  [311] = {x=105.115163, y=10.552736, z=54.518881, rx=0.000471, ry=-77.672976, rz=0.000213, shoulder=lefty, elbow=epositive, wrist=wpositive, fatherId=frmaster[1]}
  [312] = {x=103.355897, y=10.008134, z=58.376297, rx=0.003948, ry=-79.793029, rz=0.003471, shoulder=lefty, elbow=epositive, wrist=wpositive, fatherId=frmaster[1]}
  [313] = {x=101.174698, y=9.463298, z=62.618231, rx=-0.002344, ry=-82.1673, rz=-0.001686, shoulder=lefty, elbow=epositive, wrist=wpositive, fatherId=frmaster[1]}
  [314] = {x=98.49876, y=8.920808, z=67.239802, rx=-0.00454, ry=-84.819695, rz=-0.004128, shoulder=lefty, elbow=epositive, wrist=wpositive, fatherId=frmaster[1]}
  [315] = {x=95.239995, y=8.372547, z=72.223013, rx=0.011592, ry=-87.766502, rz=0.011331, shoulder=lefty, elbow=epositive, wrist=wpositive, fatherId=frmaster[1]}
  [316] = {x=93.405559, y=8.100927, z=74.780335, rx=-0.033898, ry=-89.319085, rz=-0.033723, shoulder=lefty, elbow=epositive, wrist=wpositive, fatherId=frmaster[1]}
  [317] = {x=91.396985, y=7.822504, z=77.414063, rx=-0.028938, ry=-90.956699, rz=-0.029283, shoulder=lefty, elbow=epositive, wrist=wpositive, fatherId=frmaster[1]}
  [318] = {x=89.185601, y=7.550471, z=80.130199, rx=0.005621, ry=-92.678971, rz=0.005427, shoulder=lefty, elbow=epositive, wrist=wpositive, fatherId=frmaster[1]}
  [319] = {x=86.774878, y=7.274773, z=82.909129, rx=0.003041, ry=-94.483485, rz=0.003791, shoulder=lefty, elbow=epositive, wrist=wpositive, fatherId=frmaster[1]}
  [320] = {x=84.156667, y=6.996406, z=85.721464, rx=-0.004918, ry=-96.374138, rz=-0.004959, shoulder=lefty, elbow=epositive, wrist=wpositive, fatherId=frmaster[1]}
  [321] = {x=81.287604, y=6.727029, z=88.5933, rx=0.003959, ry=-98.361433, rz=0.003574, shoulder=lefty, elbow=epositive, wrist=wpositive, fatherId=frmaster[1]}
  [322] = {x=79.766548, y=6.586584, z=90.039185, rx=0.000425, ry=-99.39159, rz=0.000719, shoulder=lefty, elbow=epositive, wrist=wpositive, fatherId=frmaster[1]}
  [323] = {x=76.689148, y=6.449037, z=92.743901, rx=-0.000115, ry=-101.368846, rz=-0.000541, shoulder=lefty, elbow=epositive, wrist=wpositive, fatherId=frmaster[1]}
  [324] = {x=72.711608, y=6.313912, z=95.955052, rx=0.002122, ry=-103.831925, rz=0.001993, shoulder=lefty, elbow=epositive, wrist=wpositive, fatherId=frmaster[1]}
  [325] = {x=68.637625, y=6.172358, z=98.971235, rx=-0.001983, ry=-106.275746, rz=-0.001913, shoulder=lefty, elbow=epositive, wrist=wpositive, fatherId=frmaster[1]}
  [326] = {x=64.204516, y=6.039868, z=101.957261, rx=0.000455, ry=-108.850801, rz=0.000254, shoulder=lefty, elbow=epositive, wrist=wpositive, fatherId=frmaster[1]}
  [327] = {x=59.531454, y=5.903167, z=104.808277, rx=-0.001203, ry=-111.487024, rz=-0.000792, shoulder=lefty, elbow=epositive, wrist=wpositive, fatherId=frmaster[1]}
  [328] = {x=54.601522, y=5.770946, z=107.502565, rx=0.000365, ry=-114.193934, rz=0.000646, shoulder=lefty, elbow=epositive, wrist=wpositive, fatherId=frmaster[1]}
  [329] = {x=49.396662, y=5.639217, z=110.0302, rx=0.001439, ry=-116.981093, rz=0.001954, shoulder=lefty, elbow=epositive, wrist=wpositive, fatherId=frmaster[1]}
  [330] = {x=43.905536, y=5.503752, z=112.367074, rx=0.001098, ry=-119.853038, rz=0.000658, shoulder=lefty, elbow=epositive, wrist=wpositive, fatherId=frmaster[1]}
  [331] = {x=38.132318, y=5.363596, z=114.489668, rx=-0.000754, ry=-122.812896, rz=-0.000603, shoulder=lefty, elbow=epositive, wrist=wpositive, fatherId=frmaster[1]}
  [332] = {x=34.633497, y=4.830797, z=115.697094, rx=-0.000999, ry=-124.728621, rz=-0.001121, shoulder=lefty, elbow=epositive, wrist=wpositive, fatherId=frmaster[1]}
  [333] = {x=32.195231, y=4.70506, z=116.424337, rx=-0.000117, ry=-125.974891, rz=-0.000379, shoulder=lefty, elbow=epositive, wrist=wpositive, fatherId=frmaster[1]}
  [334] = {x=28.076069, y=4.572613, z=117.507648, rx=0.000442, ry=-128.036025, rz=0.000186, shoulder=lefty, elbow=epositive, wrist=wpositive, fatherId=frmaster[1]}
  [335] = {x=25.057832, y=4.509903, z=118.201438, rx=0.000783, ry=-129.528131, rz=0.00073, shoulder=lefty, elbow=epositive, wrist=wpositive, fatherId=frmaster[1]}
  [336] = {x=21.435467, y=4.448246, z=118.91733, rx=0.000494, ry=-131.301627, rz=0.000656, shoulder=lefty, elbow=epositive, wrist=wpositive, fatherId=frmaster[1]}
  [337] = {x=17.185232, y=4.383492, z=119.614102, rx=0.000155, ry=-133.367865, rz=-0.000541, shoulder=lefty, elbow=epositive, wrist=wpositive, fatherId=frmaster[1]}
  [338] = {x=12.286771, y=4.319735, z=120.224792, rx=-0.000552, ry=-135.732916, rz=-0.00113, shoulder=lefty, elbow=epositive, wrist=wpositive, fatherId=frmaster[1]}
  [339] = {x=6.745577, y=4.261009, z=120.666296, rx=0.000441, ry=-138.391097, rz=-0.000116, shoulder=lefty, elbow=epositive, wrist=wpositive, fatherId=frmaster[1]}
  [340] = {x=0.626957, y=4.196667, z=120.856505, rx=-0.000387, ry=-141.317793, rz=-0.001039, shoulder=lefty, elbow=epositive, wrist=wpositive, fatherId=frmaster[1]}
  [341] = {x=-2.621994, y=4.16578, z=120.834592, rx=-0.00037, ry=-142.86837, rz=-0.000772, shoulder=lefty, elbow=epositive, wrist=wpositive, fatherId=frmaster[1]}
  [342] = {x=-8.220207, y=4.074828, z=120.570259, rx=0.000153, ry=-145.562099, rz=-0.00037, shoulder=lefty, elbow=epositive, wrist=wpositive, fatherId=frmaster[1]}
  [343] = {x=-12.173458, y=3.969382, z=120.234965, rx=-0.000075, ry=-147.496461, rz=0.000392, shoulder=lefty, elbow=epositive, wrist=wpositive, fatherId=frmaster[1]}
  [344] = {x=-16.022992, y=3.85518, z=119.762733, rx=0.000192, ry=-149.390807, rz=-0.000615, shoulder=lefty, elbow=epositive, wrist=wpositive, fatherId=frmaster[1]}
  [345] = {x=-19.771417, y=3.747011, z=119.182824, rx=0.000374, ry=-151.245321, rz=0.000006, shoulder=lefty, elbow=epositive, wrist=wpositive, fatherId=frmaster[1]}
  [346] = {x=-23.423427, y=3.639804, z=118.496959, rx=0.000566, ry=-153.06052, rz=0.000355, shoulder=lefty, elbow=epositive, wrist=wpositive, fatherId=frmaster[1]}
  [347] = {x=-27.437918, y=3.551048, z=117.608317, rx=0.000174, ry=-155.071656, rz=0.000909, shoulder=lefty, elbow=epositive, wrist=wpositive, fatherId=frmaster[1]}
  [348] = {x=-31.369091, y=3.453416, z=116.586239, rx=-0.000044, ry=-157.059735, rz=-0.000033, shoulder=lefty, elbow=epositive, wrist=wpositive, fatherId=frmaster[1]}
  [349] = {x=-35.226903, y=3.369271, z=115.441477, rx=0.000359, ry=-159.027084, rz=0.000287, shoulder=lefty, elbow=epositive, wrist=wpositive, fatherId=frmaster[1]}
  [350] = {x=-39.002937, y=3.277168, z=114.177394, rx=-0.000265, ry=-160.976303, rz=-0.000033, shoulder=lefty, elbow=epositive, wrist=wpositive, fatherId=frmaster[1]}
  [351] = {x=-43.085326, y=3.21008, z=112.652085, rx=-0.000248, ry=-163.110961, rz=0.000271, shoulder=lefty, elbow=epositive, wrist=wpositive, fatherId=frmaster[1]}
  [352] = {x=-47.122027, y=3.142962, z=110.968346, rx=0.000202, ry=-165.252195, rz=0.000493, shoulder=lefty, elbow=epositive, wrist=wpositive, fatherId=frmaster[1]}
  [353] = {x=-51.112902, y=3.070675, z=109.124081, rx=-0.00013, ry=-167.405313, rz=-0.000632, shoulder=lefty, elbow=epositive, wrist=wpositive, fatherId=frmaster[1]}
  [354] = {x=-54.974323, y=3.001944, z=107.153098, rx=0.000016, ry=-169.528533, rz=-0.000202, shoulder=lefty, elbow=epositive, wrist=wpositive, fatherId=frmaster[1]}
  [355] = {x=-59.390551, y=2.918741, z=104.602883, rx=0.000164, ry=-172.082376, rz=0.000136, shoulder=lefty, elbow=epositive, wrist=wpositive, fatherId=frmaster[1]}
  [356] = {x=-62.947412, y=2.832964, z=102.322113, rx=-0.000195, ry=-174.220706, rz=-0.000037, shoulder=lefty, elbow=epositive, wrist=wpositive, fatherId=frmaster[1]}
  [357] = {x=-62.947085, y=2.832936, z=112.317767, rx=-0.000211, ry=-174.22099, rz=0.00026, shoulder=lefty, elbow=epositive, wrist=wpositive, fatherId=frmaster[1]}
  [358] = {x=-58.458944, y=2.836341, z=156.681093, rx=0.000113, ry=-174.221159, rz=-0.000294, shoulder=lefty, elbow=epositive, wrist=wpositive, fatherId=frmaster[1]}
  [359] = {x=-18.612921, y=-20.076149, z=152.745219, rx=0.000402, ry=-174.056296, rz=-89.999944, shoulder=lefty, elbow=epositive, wrist=wpositive, fatherId=frmaster[1]}
  [360] = {x=-23.229929, y=-20.077149, z=108.388484, rx=-0.000285, ry=-174.056902, rz=-89.9999, shoulder=lefty, elbow=epositive, wrist=wpositive, fatherId=frmaster[1]}
  [361] = {x=-23.230934, y=-20.076541, z=98.391781, rx=0.000061, ry=-174.055786, rz=-89.999911, shoulder=lefty, elbow=epositive, wrist=wpositive, fatherId=frmaster[1]}
  [362] = {x=-19.340255, y=-20.472646, z=99.305974, rx=0.000015, ry=-171.571206, rz=-89.999811, shoulder=lefty, elbow=epositive, wrist=wpositive, fatherId=frmaster[1]}
  [363] = {x=-14.467347, y=-20.9313, z=100.19443, rx=179.999772, ry=-11.415156, rz=89.999471, shoulder=lefty, elbow=epositive, wrist=wpositive, fatherId=frmaster[1]}
  [364] = {x=-10.841793, y=-21.30275, z=100.675983, rx=-179.999737, ry=-13.600464, rz=89.99978, shoulder=lefty, elbow=epositive, wrist=wpositive, fatherId=frmaster[1]}
  [365] = {x=-6.648279, y=-21.675563, z=101.059651, rx=-0.000485, ry=-163.903958, rz=-89.999942, shoulder=lefty, elbow=epositive, wrist=wpositive, fatherId=frmaster[1]}
  [366] = {x=-3.944084, y=-21.97213, z=101.205494, rx=-179.999845, ry=-17.692348, rz=89.99981, shoulder=lefty, elbow=epositive, wrist=wpositive, fatherId=frmaster[1]}
  [367] = {x=-1.035961, y=-22.266805, z=101.281579, rx=0.000164, ry=-160.596349, rz=-89.999518, shoulder=lefty, elbow=epositive, wrist=wpositive, fatherId=frmaster[1]}
  [368] = {x=2.075668, y=-22.563936, z=101.263735, rx=-0.000431, ry=-158.771258, rz=-89.999398, shoulder=lefty, elbow=epositive, wrist=wpositive, fatherId=frmaster[1]}
  [369] = {x=5.374886, y=-22.856509, z=101.139982, rx=-0.00019, ry=-156.835849, rz=-89.999944, shoulder=lefty, elbow=epositive, wrist=wpositive, fatherId=frmaster[1]}
  [370] = {x=8.11646, y=-23.167098, z=100.948464, rx=179.999554, ry=-24.769598, rz=89.999348, shoulder=lefty, elbow=epositive, wrist=wpositive, fatherId=frmaster[1]}
  [371] = {x=10.839252, y=-23.473657, z=100.680376, rx=-179.999737, ry=-26.365625, rz=89.9993, shoulder=lefty, elbow=epositive, wrist=wpositive, fatherId=frmaster[1]}
  [372] = {x=14.340968, y=-24.085732, z=100.215497, rx=-179.999799, ry=-28.466933, rz=89.999508, shoulder=lefty, elbow=epositive, wrist=wpositive, fatherId=frmaster[1]}
  [373] = {x=17.063864, y=-24.631859, z=99.772139, rx=0.000249, ry=-149.886158, rz=-89.998887, shoulder=lefty, elbow=epositive, wrist=wpositive, fatherId=frmaster[1]}
  [374] = {x=19.727245, y=-25.186439, z=99.251868, rx=0.00024, ry=-148.268713, rz=-89.999973, shoulder=lefty, elbow=epositive, wrist=wpositive, fatherId=frmaster[1]}
  [375] = {x=23.493787, y=-26.015884, z=98.378332, rx=0.000126, ry=-145.960874, rz=-89.999685, shoulder=lefty, elbow=epositive, wrist=wpositive, fatherId=frmaster[1]}
  [376] = {x=27.151839, y=-26.844047, z=97.374762, rx=0.000396, ry=-143.695243, rz=-89.999786, shoulder=lefty, elbow=epositive, wrist=wpositive, fatherId=frmaster[1]}
  [377] = {x=30.702102, y=-27.677126, z=96.257879, rx=-0.001043, ry=-141.467559, rz=-89.999909, shoulder=lefty, elbow=epositive, wrist=wpositive, fatherId=frmaster[1]}
  [378] = {x=34.151197, y=-28.501632, z=95.007831, rx=0.000632, ry=-139.275172, rz=-89.999692, shoulder=lefty, elbow=epositive, wrist=wpositive, fatherId=frmaster[1]}
  [379] = {x=38.358157, y=-29.614839, z=93.291762, rx=179.999103, ry=-43.445668, rz=89.999456, shoulder=lefty, elbow=epositive, wrist=wpositive, fatherId=frmaster[1]}
  [380] = {x=40.816315, y=-30.16554, z=92.181405, rx=0.00035, ry=-134.95198, rz=-89.999842, shoulder=lefty, elbow=epositive, wrist=wpositive, fatherId=frmaster[1]}
  [381] = {x=43.623166, y=-30.723277, z=90.828073, rx=179.999263, ry=-46.887972, rz=89.999132, shoulder=lefty, elbow=epositive, wrist=wpositive, fatherId=frmaster[1]}
  [382] = {x=46.461035, y=-31.27399, z=89.349237, rx=0.000666, ry=-131.224555, rz=-89.999069, shoulder=lefty, elbow=epositive, wrist=wpositive, fatherId=frmaster[1]}
  [383] = {x=49.52499, y=-31.829878, z=87.61862, rx=0.000856, ry=-129.161053, rz=-89.998786, shoulder=lefty, elbow=epositive, wrist=wpositive, fatherId=frmaster[1]}
  [384] = {x=52.824587, y=-32.39186, z=85.592884, rx=-0.000376, ry=-126.896424, rz=-89.999824, shoulder=lefty, elbow=epositive, wrist=wpositive, fatherId=frmaster[1]}
  [385] = {x=56.368122, y=-32.945099, z=83.214974, rx=179.999887, ry=-55.592047, rz=89.99993, shoulder=lefty, elbow=epositive, wrist=wpositive, fatherId=frmaster[1]}
  [386] = {x=59.982794, y=-33.501646, z=80.56291, rx=0.000356, ry=-121.795353, rz=-89.999372, shoulder=lefty, elbow=epositive, wrist=wpositive, fatherId=frmaster[1]}
  [387] = {x=63.860131, y=-34.057469, z=77.43317, rx=0.001113, ry=-118.892986, rz=-89.998492, shoulder=lefty, elbow=epositive, wrist=wpositive, fatherId=frmaster[1]}
  [388] = {x=65.894571, y=-34.341079, z=75.654242, rx=179.999036, ry=-62.672719, rz=89.998766, shoulder=lefty, elbow=epositive, wrist=wpositive, fatherId=frmaster[1]}
  [389] = {x=67.978967, y=-34.617239, z=73.736742, rx=0.000688, ry=-115.679952, rz=-89.998265, shoulder=lefty, elbow=epositive, wrist=wpositive, fatherId=frmaster[1]}
  [390] = {x=70.113955, y=-34.895869, z=71.65174, rx=179.999274, ry=-66.045856, rz=89.999704, shoulder=lefty, elbow=epositive, wrist=wpositive, fatherId=frmaster[1]}
  [391] = {x=72.277536, y=-35.178962, z=69.406219, rx=179.998605, ry=-67.852148, rz=89.998988, shoulder=lefty, elbow=epositive, wrist=wpositive, fatherId=frmaster[1]}
  [392] = {x=74.376116, y=-35.45348, z=67.085303, rx=179.999869, ry=-69.662949, rz=89.999758, shoulder=lefty, elbow=epositive, wrist=wpositive, fatherId=frmaster[1]}
  [393] = {x=76.513977, y=-35.730157, z=64.566903, rx=0.000592, ry=-108.424559, rz=-89.999536, shoulder=lefty, elbow=epositive, wrist=wpositive, fatherId=frmaster[1]}
  [394] = {x=78.679667, y=-36.009316, z=61.843135, rx=0.001385, ry=-106.410069, rz=-89.998392, shoulder=lefty, elbow=epositive, wrist=wpositive, fatherId=frmaster[1]}
  [395] = {x=80.846119, y=-36.288822, z=58.903263, rx=0.000878, ry=-104.297201, rz=-89.999128, shoulder=lefty, elbow=epositive, wrist=wpositive, fatherId=frmaster[1]}
  [396] = {x=82.995135, y=-36.570009, z=55.747917, rx=179.999305, ry=-77.907489, rz=89.999806, shoulder=lefty, elbow=epositive, wrist=wpositive, fatherId=frmaster[1]}
  [397] = {x=85.094465, y=-36.847128, z=52.391805, rx=0.001232, ry=-99.802552, rz=-89.998506, shoulder=lefty, elbow=epositive, wrist=wpositive, fatherId=frmaster[1]}
  [398] = {x=87.124675, y=-37.127203, z=48.843094, rx=0.000325, ry=-97.44439, rz=-89.999996, shoulder=lefty, elbow=epositive, wrist=wpositive, fatherId=frmaster[1]}
  [399] = {x=89.220179, y=-37.40856, z=44.781627, rx=179.996062, ry=-85.19367, rz=89.995853, shoulder=lefty, elbow=epositive, wrist=wpositive, fatherId=frmaster[1]}
  [400] = {x=90.407375, y=-37.548857, z=42.270351, rx=0.000347, ry=-93.204424, rz=-89.999876, shoulder=lefty, elbow=epositive, wrist=wpositive, fatherId=frmaster[1]}
  [401] = {x=91.449184, y=-37.685314, z=39.897994, rx=179.994643, ry=-88.288606, rz=89.994157, shoulder=lefty, elbow=epositive, wrist=wpositive, fatherId=frmaster[1]}
  [402] = {x=93.126378, y=-37.965093, z=35.654137, rx=-0.009346, ry=-89.071193, rz=-90.008547, shoulder=lefty, elbow=epositive, wrist=wpositive, fatherId=frmaster[1]}
  [403] = {x=94.341626, y=-38.242334, z=32.113083, rx=-0.002381, ry=-86.91033, rz=-90.002294, shoulder=lefty, elbow=epositive, wrist=wpositive, fatherId=frmaster[1]}
  [404] = {x=95.188068, y=-38.521496, z=29.326357, rx=-0.006605, ry=-85.224912, rz=-90.006769, shoulder=lefty, elbow=epositive, wrist=wpositive, fatherId=frmaster[1]}
  [405] = {x=96.037478, y=-39.643639, z=25.537786, rx=0.005745, ry=-82.953272, rz=-89.993502, shoulder=lefty, elbow=epositive, wrist=wpositive, fatherId=frmaster[1]}
  [406] = {x=96.050516, y=-41.866509, z=23.488772, rx=0.004459, ry=-81.734218, rz=-89.996102, shoulder=lefty, elbow=epositive, wrist=wpositive, fatherId=frmaster[1]}
  [407] = {x=96.265179, y=-44.084468, z=20.099386, rx=0.001458, ry=-79.713403, rz=-89.998028, shoulder=lefty, elbow=epositive, wrist=wpositive, fatherId=frmaster[1]}
  [408] = {x=95.830359, y=-46.300323, z=19.531156, rx=-0.000494, ry=-79.37359, rz=-89.999699, shoulder=lefty, elbow=epositive, wrist=wpositive, fatherId=frmaster[1]}
  [409] = {x=95.219744, y=-48.498071, z=19.530741, rx=-0.001577, ry=-79.373839, rz=-90.00152, shoulder=lefty, elbow=epositive, wrist=wpositive, fatherId=frmaster[1]}
  [410] = {x=94.610866, y=-50.699727, z=19.525133, rx=-0.00248, ry=-79.37452, rz=-90.0025, shoulder=lefty, elbow=epositive, wrist=wpositive, fatherId=frmaster[1]}
  [411] = {x=93.949121, y=-52.887868, z=19.527792, rx=0.000679, ry=-79.373805, rz=-89.999525, shoulder=lefty, elbow=epositive, wrist=wpositive, fatherId=frmaster[1]}
  [412] = {x=93.291001, y=-55.07631, z=19.529205, rx=-0.000585, ry=-79.373856, rz=-89.999996, shoulder=lefty, elbow=epositive, wrist=wpositive, fatherId=frmaster[1]}
  [413] = {x=92.575078, y=-57.243716, z=19.530074, rx=0.000066, ry=-79.374019, rz=-89.999528, shoulder=lefty, elbow=epositive, wrist=wpositive, fatherId=frmaster[1]}
  [414] = {x=91.860687, y=-59.413792, z=19.526132, rx=0.001303, ry=-79.374478, rz=-89.99887, shoulder=lefty, elbow=epositive, wrist=wpositive, fatherId=frmaster[1]}
  [415] = {x=91.092576, y=-61.567574, z=19.530938, rx=0.002328, ry=-79.373689, rz=-89.997279, shoulder=lefty, elbow=epositive, wrist=wpositive, fatherId=frmaster[1]}
  [416] = {x=90.320474, y=-63.717023, z=19.531145, rx=-0.001214, ry=-79.373131, rz=-90.000771, shoulder=lefty, elbow=epositive, wrist=wpositive, fatherId=frmaster[1]}
  [417] = {x=91.145025, y=-61.620795, z=19.526573, rx=0.003847, ry=-79.373786, rz=-89.996531, shoulder=lefty, elbow=epositive, wrist=wpositive, fatherId=frmaster[1]}
  [418] = {x=91.960756, y=-59.522744, z=19.529359, rx=-0.001864, ry=-79.37355, rz=-90.001891, shoulder=lefty, elbow=epositive, wrist=wpositive, fatherId=frmaster[1]}
  [419] = {x=92.778954, y=-57.426276, z=19.531234, rx=0.000056, ry=-79.373948, rz=-89.999483, shoulder=lefty, elbow=epositive, wrist=wpositive, fatherId=frmaster[1]}
  [420] = {x=93.363053, y=-55.842732, z=19.529047, rx=0.003047, ry=-79.373636, rz=-89.996853, shoulder=lefty, elbow=epositive, wrist=wpositive, fatherId=frmaster[1]}
  [421] = {x=93.94496, y=-54.257234, z=19.527324, rx=0.001148, ry=-79.374432, rz=-89.998674, shoulder=lefty, elbow=epositive, wrist=wpositive, fatherId=frmaster[1]}
  [422] = {x=94.48512, y=-52.658764, z=19.530193, rx=-0.001331, ry=-79.373615, rz=-90.001137, shoulder=lefty, elbow=epositive, wrist=wpositive, fatherId=frmaster[1]}
  [423] = {x=95.029562, y=-51.065002, z=19.525702, rx=0.001956, ry=-79.374266, rz=-89.99832, shoulder=lefty, elbow=epositive, wrist=wpositive, fatherId=frmaster[1]}
  [424] = {x=95.510279, y=-49.447929, z=19.531705, rx=-0.003616, ry=-79.373366, rz=-90.003709, shoulder=lefty, elbow=epositive, wrist=wpositive, fatherId=frmaster[1]}
  [425] = {x=95.998787, y=-47.833562, z=19.527851, rx=-0.000252, ry=-79.373407, rz=-90.00061, shoulder=lefty, elbow=epositive, wrist=wpositive, fatherId=frmaster[1]}
  [426] = {x=96.179927, y=-45.385772, z=21.661715, rx=-0.000722, ry=-80.643878, rz=-90.000709, shoulder=lefty, elbow=epositive, wrist=wpositive, fatherId=frmaster[1]}
  [427] = {x=96.007005, y=-43.535446, z=23.987198, rx=0.003627, ry=-82.030083, rz=-89.996774, shoulder=lefty, elbow=epositive, wrist=wpositive, fatherId=frmaster[1]}
  [428] = {x=95.813262, y=-41.683229, z=26.194793, rx=0.000832, ry=-83.349603, rz=-89.999368, shoulder=lefty, elbow=epositive, wrist=wpositive, fatherId=frmaster[1]}
  [429] = {x=95.286759, y=-39.809655, z=28.973952, rx=0.002677, ry=-85.016425, rz=-89.997383, shoulder=lefty, elbow=epositive, wrist=wpositive, fatherId=frmaster[1]}
  [430] = {x=93.741309, y=-38.868588, z=33.91884, rx=-0.005481, ry=-88.010972, rz=-90.005409, shoulder=lefty, elbow=epositive, wrist=wpositive, fatherId=frmaster[1]}
  [431] = {x=92.557837, y=-38.404543, z=37.167212, rx=177.137756, ry=-89.993959, rz=87.137837, shoulder=lefty, elbow=epositive, wrist=wpositive, fatherId=frmaster[1]}
  [432] = {x=91.030198, y=-37.932071, z=40.88008, rx=179.995934, ry=-87.675502, rz=89.99589, shoulder=lefty, elbow=epositive, wrist=wpositive, fatherId=frmaster[1]}
  [433] = {x=89.692317, y=-37.097359, z=43.80771, rx=179.998028, ry=-85.81607, rz=89.997801, shoulder=lefty, elbow=epositive, wrist=wpositive, fatherId=frmaster[1]}
  [434] = {x=88.245296, y=-36.25766, z=46.717015, rx=0.000432, ry=-96.055165, rz=-89.999914, shoulder=lefty, elbow=epositive, wrist=wpositive, fatherId=frmaster[1]}
  [435] = {x=85.834088, y=-34.585456, z=51.131918, rx=0.001437, ry=-98.96274, rz=-89.998711, shoulder=lefty, elbow=epositive, wrist=wpositive, fatherId=frmaster[1]}
  [436] = {x=87.363997, y=-33.334451, z=48.399633, rx=179.997154, ry=-82.850828, rz=89.997631, shoulder=lefty, elbow=epositive, wrist=wpositive, fatherId=frmaster[1]}
  [437] = {x=88.963104, y=-32.078964, z=45.308637, rx=179.998939, ry=-84.858105, rz=89.999166, shoulder=lefty, elbow=epositive, wrist=wpositive, fatherId=frmaster[1]}
  [438] = {x=90.833345, y=-31.60392, z=41.317379, rx=0.014923, ry=-92.601946, rz=-89.985219, shoulder=lefty, elbow=epositive, wrist=wpositive, fatherId=frmaster[1]}
  [439] = {x=92.343037, y=-31.135471, z=37.709578, rx=0.079131, ry=-90.34356, rz=-89.920987, shoulder=lefty, elbow=epositive, wrist=wpositive, fatherId=frmaster[1]}
  [440] = {x=93.529677, y=-30.666154, z=34.531814, rx=-0.017187, ry=-88.384847, rz=-90.017514, shoulder=lefty, elbow=epositive, wrist=wpositive, fatherId=frmaster[1]}
  [441] = {x=94.442975, y=-30.199384, z=31.814924, rx=0.010171, ry=-86.731017, rz=-89.990611, shoulder=lefty, elbow=epositive, wrist=wpositive, fatherId=frmaster[1]}
  [442] = {x=95.823658, y=-29.50404, z=26.92009, rx=0.002771, ry=-83.781123, rz=-89.997667, shoulder=lefty, elbow=epositive, wrist=wpositive, fatherId=frmaster[1]}
  [443] = {x=95.887318, y=-27.417283, z=25.270326, rx=-0.004655, ry=-82.794198, rz=-90.004079, shoulder=lefty, elbow=epositive, wrist=wpositive, fatherId=frmaster[1]}
  [444] = {x=96.236472, y=-24.692541, z=20.696818, rx=0.003439, ry=-80.067759, rz=-89.996112, shoulder=lefty, elbow=epositive, wrist=wpositive, fatherId=frmaster[1]}
  [445] = {x=95.914737, y=-23.107464, z=19.528885, rx=-0.000161, ry=-79.373394, rz=-90.000119, shoulder=lefty, elbow=epositive, wrist=wpositive, fatherId=frmaster[1]}
  [446] = {x=95.348602, y=-21.519123, z=19.529286, rx=0.000907, ry=-79.373786, rz=-89.999424, shoulder=lefty, elbow=epositive, wrist=wpositive, fatherId=frmaster[1]}
  [447] = {x=94.371853, y=-19.183629, z=19.524151, rx=-0.001736, ry=-79.374377, rz=-90.002228, shoulder=lefty, elbow=epositive, wrist=wpositive, fatherId=frmaster[1]}
  [448] = {x=93.316622, y=-16.883116, z=19.526275, rx=0.000956, ry=-79.374307, rz=-89.999709, shoulder=lefty, elbow=epositive, wrist=wpositive, fatherId=frmaster[1]}
  [449] = {x=92.223198, y=-14.597643, z=19.527179, rx=-0.002205, ry=-79.374225, rz=-90.002362, shoulder=lefty, elbow=epositive, wrist=wpositive, fatherId=frmaster[1]}
  [450] = {x=91.132258, y=-12.322218, z=19.528965, rx=0.000461, ry=-79.374174, rz=-89.999351, shoulder=lefty, elbow=epositive, wrist=wpositive, fatherId=frmaster[1]}
  [451] = {x=90.438196, y=-10.806794, z=19.525651, rx=-0.001834, ry=-79.374261, rz=-90.002371, shoulder=lefty, elbow=epositive, wrist=wpositive, fatherId=frmaster[1]}
  [452] = {x=89.748446, y=-9.293815, z=19.525833, rx=0.000667, ry=-79.374008, rz=-89.999146, shoulder=lefty, elbow=epositive, wrist=wpositive, fatherId=frmaster[1]}
  [453] = {x=89.128569, y=-7.746741, z=19.526477, rx=-0.000458, ry=-79.374167, rz=-90.000826, shoulder=lefty, elbow=epositive, wrist=wpositive, fatherId=frmaster[1]}
  [454] = {x=88.513421, y=-6.201062, z=19.531404, rx=-0.003371, ry=-79.373381, rz=-90.003437, shoulder=lefty, elbow=epositive, wrist=wpositive, fatherId=frmaster[1]}
  [455] = {x=87.987684, y=-4.643, z=19.529166, rx=-0.004354, ry=-79.37384, rz=-90.004523, shoulder=lefty, elbow=epositive, wrist=wpositive, fatherId=frmaster[1]}
  [456] = {x=87.538091, y=-3.067935, z=19.531336, rx=0.001659, ry=-79.374002, rz=-89.997873, shoulder=lefty, elbow=epositive, wrist=wpositive, fatherId=frmaster[1]}
  [457] = {x=87.169272, y=-1.461613, z=19.525964, rx=0.001276, ry=-79.373742, rz=-89.999306, shoulder=lefty, elbow=epositive, wrist=wpositive, fatherId=frmaster[1]}
  [458] = {x=86.898988, y=0.152966, z=19.530489, rx=0.001657, ry=-79.373367, rz=-89.998042, shoulder=lefty, elbow=epositive, wrist=wpositive, fatherId=frmaster[1]}
  [459] = {x=86.740855, y=1.80285, z=19.527201, rx=0.001016, ry=-79.374209, rz=-89.999139, shoulder=lefty, elbow=epositive, wrist=wpositive, fatherId=frmaster[1]}
  [460] = {x=86.71752, y=3.243751, z=19.530114, rx=-0.0037, ry=-79.374292, rz=-90.004085, shoulder=lefty, elbow=epositive, wrist=wpositive, fatherId=frmaster[1]}
  [461] = {x=86.796381, y=4.677729, z=19.529878, rx=-0.004118, ry=-79.373247, rz=-90.003724, shoulder=lefty, elbow=epositive, wrist=wpositive, fatherId=frmaster[1]}
  [462] = {x=87.094524, y=6.831768, z=19.532133, rx=-0.000159, ry=-79.373041, rz=-90.000065, shoulder=lefty, elbow=epositive, wrist=wpositive, fatherId=frmaster[1]}
  [463] = {x=87.574161, y=8.955411, z=19.531743, rx=0.001046, ry=-79.373481, rz=-89.998729, shoulder=lefty, elbow=epositive, wrist=wpositive, fatherId=frmaster[1]}
  [464] = {x=88.199153, y=11.055864, z=19.526103, rx=-0.003033, ry=-79.374007, rz=-90.002836, shoulder=lefty, elbow=epositive, wrist=wpositive, fatherId=frmaster[1]}
  [465] = {x=88.93354, y=13.104978, z=19.530227, rx=-0.002055, ry=-79.373473, rz=-90.001816, shoulder=lefty, elbow=epositive, wrist=wpositive, fatherId=frmaster[1]}
  [466] = {x=89.580648, y=14.657762, z=19.527802, rx=-0.004099, ry=-79.373793, rz=-90.003771, shoulder=lefty, elbow=epositive, wrist=wpositive, fatherId=frmaster[1]}
  [467] = {x=90.229958, y=16.20197, z=19.527384, rx=0.001444, ry=-79.373644, rz=-89.998136, shoulder=lefty, elbow=epositive, wrist=wpositive, fatherId=frmaster[1]}
  [468] = {x=90.932763, y=17.729652, z=19.527434, rx=-0.000339, ry=-79.373536, rz=-90.000584, shoulder=lefty, elbow=epositive, wrist=wpositive, fatherId=frmaster[1]}
  [469] = {x=91.633231, y=19.254728, z=19.528456, rx=0.00169, ry=-79.37389, rz=-89.998345, shoulder=lefty, elbow=epositive, wrist=wpositive, fatherId=frmaster[1]}
  [470] = {x=92.346151, y=20.773499, z=19.533352, rx=-0.001041, ry=-79.373453, rz=-90.000406, shoulder=lefty, elbow=epositive, wrist=wpositive, fatherId=frmaster[1]}
  [471] = {x=93.061959, y=22.293661, z=19.530607, rx=-0.001807, ry=-79.373187, rz=-90.001727, shoulder=lefty, elbow=epositive, wrist=wpositive, fatherId=frmaster[1]}
  [472] = {x=93.749131, y=23.815646, z=19.532795, rx=0.003181, ry=-79.373036, rz=-89.996919, shoulder=lefty, elbow=epositive, wrist=wpositive, fatherId=frmaster[1]}
  [473] = {x=94.435063, y=25.345879, z=19.525859, rx=0.001086, ry=-79.374317, rz=-89.999214, shoulder=lefty, elbow=epositive, wrist=wpositive, fatherId=frmaster[1]}
  [474] = {x=95.056156, y=26.892076, z=19.525042, rx=-0.000444, ry=-79.374189, rz=-90.00051, shoulder=lefty, elbow=epositive, wrist=wpositive, fatherId=frmaster[1]}
  [475] = {x=95.67128, y=28.440192, z=19.525181, rx=0.001353, ry=-79.374346, rz=-89.998934, shoulder=lefty, elbow=epositive, wrist=wpositive, fatherId=frmaster[1]}
  [476] = {x=96.177659, y=30.02891, z=19.530228, rx=-0.004211, ry=-79.373309, rz=-90.003725, shoulder=lefty, elbow=epositive, wrist=wpositive, fatherId=frmaster[1]}
  [477] = {x=96.159546, y=31.608712, z=21.97677, rx=0.004599, ry=-80.828096, rz=-89.995097, shoulder=lefty, elbow=epositive, wrist=wpositive, fatherId=frmaster[1]}
  [478] = {x=95.972967, y=33.233743, z=24.387706, rx=0.000185, ry=-82.269693, rz=-89.999554, shoulder=lefty, elbow=epositive, wrist=wpositive, fatherId=frmaster[1]}
  [479] = {x=96.120098, y=35.695229, z=25.361113, rx=0.004034, ry=-82.852647, rz=-89.996529, shoulder=lefty, elbow=epositive, wrist=wpositive, fatherId=frmaster[1]}
  [480] = {x=95.464563, y=38.187701, z=28.332828, rx=0.002269, ry=-84.63219, rz=-89.997812, shoulder=lefty, elbow=epositive, wrist=wpositive, fatherId=frmaster[1]}
  [481] = {x=95.481944, y=39.857513, z=28.262466, rx=-0.005347, ry=-84.586394, rz=-90.005308, shoulder=lefty, elbow=epositive, wrist=wpositive, fatherId=frmaster[1]}
  [482] = {x=96.046267, y=41.521619, z=25.932821, rx=-0.005246, ry=-83.190222, rz=-90.005051, shoulder=lefty, elbow=epositive, wrist=wpositive, fatherId=frmaster[1]}
  [483] = {x=95.867169, y=44.008908, z=25.453729, rx=-0.005438, ry=-82.902776, rz=-90.004534, shoulder=lefty, elbow=epositive, wrist=wpositive, fatherId=frmaster[1]}
  [484] = {x=96.060662, y=45.848865, z=23.368454, rx=0.003558, ry=-81.661301, rz=-89.996621, shoulder=lefty, elbow=epositive, wrist=wpositive, fatherId=frmaster[1]}
  [485] = {x=96.231426, y=47.678688, z=20.770954, rx=-0.001012, ry=-80.114502, rz=-90.001398, shoulder=lefty, elbow=epositive, wrist=wpositive, fatherId=frmaster[1]}
  [486] = {x=95.960361, y=49.475692, z=19.529546, rx=-0.003131, ry=-79.37362, rz=-90.002756, shoulder=lefty, elbow=epositive, wrist=wpositive, fatherId=frmaster[1]}
  [487] = {x=95.435065, y=51.270997, z=19.528082, rx=0.002665, ry=-79.373716, rz=-89.997938, shoulder=lefty, elbow=epositive, wrist=wpositive, fatherId=frmaster[1]}
  [488] = {x=94.862455, y=52.855164, z=19.530682, rx=0.000492, ry=-79.373096, rz=-89.999094, shoulder=lefty, elbow=epositive, wrist=wpositive, fatherId=frmaster[1]}
  [489] = {x=94.295363, y=54.438366, z=19.527634, rx=-0.000115, ry=-79.374198, rz=-90.000488, shoulder=lefty, elbow=epositive, wrist=wpositive, fatherId=frmaster[1]}
  [490] = {x=93.662758, y=55.991812, z=19.531446, rx=0.002594, ry=-79.373106, rz=-89.997131, shoulder=lefty, elbow=epositive, wrist=wpositive, fatherId=frmaster[1]}
  [491] = {x=93.031933, y=57.551191, z=19.529577, rx=0.001381, ry=-79.373693, rz=-89.998678, shoulder=lefty, elbow=epositive, wrist=wpositive, fatherId=frmaster[1]}
  [492] = {x=92.130556, y=59.608746, z=19.526668, rx=0.001831, ry=-79.373665, rz=-89.99885, shoulder=lefty, elbow=epositive, wrist=wpositive, fatherId=frmaster[1]}
  [493] = {x=91.227931, y=61.660848, z=19.526186, rx=0.003295, ry=-79.374183, rz=-89.996436, shoulder=lefty, elbow=epositive, wrist=wpositive, fatherId=frmaster[1]}
  [494] = {x=90.325218, y=63.715632, z=19.527445, rx=0.003861, ry=-79.373934, rz=-89.996204, shoulder=lefty, elbow=epositive, wrist=wpositive, fatherId=frmaster[1]}
  [495] = {x=91.090514, y=61.562981, z=19.529622, rx=-0.001852, ry=-79.37323, rz=-90.001702, shoulder=lefty, elbow=epositive, wrist=wpositive, fatherId=frmaster[1]}
  [496] = {x=91.860274, y=59.404675, z=19.532383, rx=-0.001616, ry=-79.372906, rz=-90.001198, shoulder=lefty, elbow=epositive, wrist=wpositive, fatherId=frmaster[1]}
  [497] = {x=92.577582, y=57.228632, z=19.528048, rx=0.003602, ry=-79.373353, rz=-89.996066, shoulder=lefty, elbow=epositive, wrist=wpositive, fatherId=frmaster[1]}
  [498] = {x=93.291801, y=55.05905, z=19.531235, rx=-0.00138, ry=-79.373582, rz=-90.001363, shoulder=lefty, elbow=epositive, wrist=wpositive, fatherId=frmaster[1]}
  [499] = {x=93.954362, y=52.870428, z=19.528627, rx=-0.002203, ry=-79.373694, rz=-90.002633, shoulder=lefty, elbow=epositive, wrist=wpositive, fatherId=frmaster[1]}
  [500] = {x=94.6188, y=50.680643, z=19.52677, rx=-0.001982, ry=-79.374301, rz=-90.002654, shoulder=lefty, elbow=epositive, wrist=wpositive, fatherId=frmaster[1]}
  [501] = {x=95.231085, y=48.469644, z=19.526413, rx=0.002198, ry=-79.374018, rz=-89.998138, shoulder=lefty, elbow=epositive, wrist=wpositive, fatherId=frmaster[1]}
  [502] = {x=95.838547, y=46.269084, z=19.52693, rx=-0.003028, ry=-79.37429, rz=-90.002888, shoulder=lefty, elbow=epositive, wrist=wpositive, fatherId=frmaster[1]}
  [503] = {x=96.259771, y=44.048497, z=20.156876, rx=-0.000308, ry=-79.747784, rz=-90.000296, shoulder=lefty, elbow=epositive, wrist=wpositive, fatherId=frmaster[1]}
  [504] = {x=96.043978, y=41.828635, z=23.543569, rx=-0.002072, ry=-81.767601, rz=-90.002394, shoulder=lefty, elbow=epositive, wrist=wpositive, fatherId=frmaster[1]}
  [505] = {x=96.063412, y=39.595477, z=25.464842, rx=-0.00122, ry=-82.913981, rz=-90.000898, shoulder=lefty, elbow=epositive, wrist=wpositive, fatherId=frmaster[1]}
  [506] = {x=95.073024, y=38.479974, z=29.732493, rx=-0.001761, ry=-85.470976, rz=-90.002172, shoulder=lefty, elbow=epositive, wrist=wpositive, fatherId=frmaster[1]}
  [507] = {x=94.171412, y=38.194631, z=32.650909, rx=0.009411, ry=-87.235053, rz=-89.990645, shoulder=lefty, elbow=epositive, wrist=wpositive, fatherId=frmaster[1]}
  [508] = {x=92.885211, y=37.921331, z=36.301375, rx=-0.059985, ry=-89.473319, rz=-90.060282, shoulder=lefty, elbow=epositive, wrist=wpositive, fatherId=frmaster[1]}
  [509] = {x=91.131904, y=37.637999, z=40.64419, rx=0.000556, ry=-92.178714, rz=-89.999837, shoulder=lefty, elbow=epositive, wrist=wpositive, fatherId=frmaster[1]}
  [510] = {x=90.053254, y=37.498763, z=43.044666, rx=179.998068, ry=-86.302008, rz=89.997341, shoulder=lefty, elbow=epositive, wrist=wpositive, fatherId=frmaster[1]}
  [511] = {x=88.829752, y=37.358252, z=45.57431, rx=179.994876, ry=-84.681965, rz=89.993899, shoulder=lefty, elbow=epositive, wrist=wpositive, fatherId=frmaster[1]}
  [512] = {x=86.811968, y=37.079632, z=49.413338, rx=179.998796, ry=-82.180427, rz=89.998382, shoulder=lefty, elbow=epositive, wrist=wpositive, fatherId=frmaster[1]}
  [513] = {x=84.768484, y=36.795715, z=52.935938, rx=179.997667, ry=-79.829512, rz=89.99811, shoulder=lefty, elbow=epositive, wrist=wpositive, fatherId=frmaster[1]}
  [514] = {x=82.64898, y=36.516486, z=56.277671, rx=179.997601, ry=-77.544884, rz=89.998328, shoulder=lefty, elbow=epositive, wrist=wpositive, fatherId=frmaster[1]}
  [515] = {x=80.483198, y=36.244003, z=59.406943, rx=0.002512, ry=-104.660347, rz=-89.997714, shoulder=lefty, elbow=epositive, wrist=wpositive, fatherId=frmaster[1]}
  [516] = {x=78.298826, y=35.958402, z=62.341358, rx=179.999209, ry=-73.227242, rz=89.999295, shoulder=lefty, elbow=epositive, wrist=wpositive, fatherId=frmaster[1]}
  [517] = {x=76.116113, y=35.677941, z=65.053942, rx=179.999239, ry=-71.209576, rz=89.998848, shoulder=lefty, elbow=epositive, wrist=wpositive, fatherId=frmaster[1]}
  [518] = {x=73.953097, y=35.400213, z=67.564566, rx=0.00063, ry=-110.707071, rz=-89.999417, shoulder=lefty, elbow=epositive, wrist=wpositive, fatherId=frmaster[1]}
  [519] = {x=71.832107, y=35.12216, z=69.876286, rx=0.001182, ry=-112.522933, rz=-89.999536, shoulder=lefty, elbow=epositive, wrist=wpositive, fatherId=frmaster[1]}
  [520] = {x=69.662712, y=34.838948, z=72.101404, rx=179.999465, ry=-65.67559, rz=89.999123, shoulder=lefty, elbow=epositive, wrist=wpositive, fatherId=frmaster[1]}
  [521] = {x=67.521312, y=34.560084, z=74.170278, rx=179.999605, ry=-63.954773, rz=89.999652, shoulder=lefty, elbow=epositive, wrist=wpositive, fatherId=frmaster[1]}
  [522] = {x=65.431652, y=34.278654, z=76.069471, rx=179.998956, ry=-62.312584, rz=89.998714, shoulder=lefty, elbow=epositive, wrist=wpositive, fatherId=frmaster[1]}
  [523] = {x=63.39483, y=34.001592, z=77.828634, rx=0.000514, ry=-119.247856, rz=-89.998951, shoulder=lefty, elbow=epositive, wrist=wpositive, fatherId=frmaster[1]}
  [524] = {x=59.51443, y=33.440695, z=80.92467, rx=179.999467, ry=-57.860726, rz=89.999379, shoulder=lefty, elbow=epositive, wrist=wpositive, fatherId=frmaster[1]}
  [525] = {x=55.896957, y=32.881756, z=83.548671, rx=179.999387, ry=-55.258926, rz=89.99943, shoulder=lefty, elbow=epositive, wrist=wpositive, fatherId=frmaster[1]}
  [526] = {x=52.333231, y=32.328266, z=85.902825, rx=0.000304, ry=-127.235919, rz=-89.998732, shoulder=lefty, elbow=epositive, wrist=wpositive, fatherId=frmaster[1]}
  [527] = {x=49.0222, y=31.768772, z=87.904906, rx=0.00109, ry=-129.505408, rz=-89.999155, shoulder=lefty, elbow=epositive, wrist=wpositive, fatherId=frmaster[1]}
  [528] = {x=45.94524, y=31.208896, z=89.622718, rx=179.999556, ry=-48.427884, rz=89.999581, shoulder=lefty, elbow=epositive, wrist=wpositive, fatherId=frmaster[1]}
  [529] = {x=43.089364, y=30.651004, z=91.093136, rx=-179.999993, ry=-46.537967, rz=89.999814, shoulder=lefty, elbow=epositive, wrist=wpositive, fatherId=frmaster[1]}
  [530] = {x=40.3343, y=30.094346, z=92.41051, rx=0.000233, ry=-135.265763, rz=-89.999307, shoulder=lefty, elbow=epositive, wrist=wpositive, fatherId=frmaster[1]}
  [531] = {x=38.000421, y=29.534038, z=93.443046, rx=179.999339, ry=-43.210248, rz=89.99887, shoulder=lefty, elbow=epositive, wrist=wpositive, fatherId=frmaster[1]}
  [532] = {x=33.813267, y=28.42418, z=95.138765, rx=0.000803, ry=-139.491071, rz=-89.999251, shoulder=lefty, elbow=epositive, wrist=wpositive, fatherId=frmaster[1]}
  [533] = {x=29.279696, y=27.311224, z=96.723566, rx=179.999493, ry=-37.634598, rz=89.99936, shoulder=lefty, elbow=epositive, wrist=wpositive, fatherId=frmaster[1]}
  [534] = {x=24.57798, y=26.204339, z=98.101157, rx=0.000526, ry=-145.29105, rz=-89.999557, shoulder=lefty, elbow=epositive, wrist=wpositive, fatherId=frmaster[1]}
  [535] = {x=21.948268, y=25.650271, z=98.755366, rx=-179.999904, ry=-33.089678, rz=89.999844, shoulder=lefty, elbow=epositive, wrist=wpositive, fatherId=frmaster[1]}
  [536] = {x=19.252704, y=25.096926, z=99.348172, rx=-179.999779, ry=-31.440758, rz=89.999431, shoulder=lefty, elbow=epositive, wrist=wpositive, fatherId=frmaster[1]}
  [537] = {x=16.482905, y=24.549838, z=99.868502, rx=0.000162, ry=-150.238919, rz=-89.999206, shoulder=lefty, elbow=epositive, wrist=wpositive, fatherId=frmaster[1]}
  [538] = {x=13.644071, y=23.996072, z=100.321389, rx=0.000105, ry=-151.94971, rz=-89.999728, shoulder=lefty, elbow=epositive, wrist=wpositive, fatherId=frmaster[1]}
  [539] = {x=10.533698, y=23.4521, z=100.717783, rx=179.999742, ry=-26.185436, rz=89.998948, shoulder=lefty, elbow=epositive, wrist=wpositive, fatherId=frmaster[1]}
  [540] = {x=5.632137, y=22.912745, z=101.123848, rx=179.999896, ry=-23.314365, rz=89.999698, shoulder=lefty, elbow=epositive, wrist=wpositive, fatherId=frmaster[1]}
  [541] = {x=2.843467, y=22.648765, z=101.241436, rx=0.000638, ry=-158.320888, rz=-89.999767, shoulder=lefty, elbow=epositive, wrist=wpositive, fatherId=frmaster[1]}
  [542] = {x=0.189441, y=22.376516, z=101.283624, rx=-0.000269, ry=-159.875907, rz=-89.999649, shoulder=lefty, elbow=epositive, wrist=wpositive, fatherId=frmaster[1]}
  [543] = {x=-4.685542, y=21.843586, z=101.171838, rx=-0.000226, ry=-162.743918, rz=-89.999173, shoulder=lefty, elbow=epositive, wrist=wpositive, fatherId=frmaster[1]}
  [544] = {x=-7.646892, y=21.596476, z=100.983437, rx=-179.999729, ry=-15.50282, rz=89.99972, shoulder=lefty, elbow=epositive, wrist=wpositive, fatherId=frmaster[1]}
  [545] = {x=-10.363278, y=21.345744, z=100.723264, rx=-179.999638, ry=-13.882905, rz=89.999535, shoulder=lefty, elbow=epositive, wrist=wpositive, fatherId=frmaster[1]}
  [546] = {x=-15.082995, y=20.854317, z=100.093618, rx=-179.999828, ry=-11.043003, rz=89.999638, shoulder=lefty, elbow=epositive, wrist=wpositive, fatherId=frmaster[1]}
  [547] = {x=-19.817489, y=20.42773, z=99.211625, rx=-0.000037, ry=-171.869727, rz=-89.99931, shoulder=lefty, elbow=epositive, wrist=wpositive, fatherId=frmaster[1]}
  [548] = {x=-23.463327, y=20.052779, z=98.325324, rx=0.000305, ry=-174.211932, rz=-89.999824, shoulder=lefty, elbow=epositive, wrist=wpositive, fatherId=frmaster[1]}
  [549] = {x=-23.463042, y=20.052956, z=108.316879, rx=0.00049, ry=-174.212256, rz=-89.999952, shoulder=lefty, elbow=epositive, wrist=wpositive, fatherId=frmaster[1]}
  [550] = {x=-18.965231, y=20.04784, z=152.690581, rx=-0.000036, ry=-174.211316, rz=-89.999767, shoulder=lefty, elbow=epositive, wrist=wpositive, fatherId=frmaster[1]}
  [551] = {x=-58.457155, y=-2.837264, z=156.675838, rx=-179.999805, ry=-5.778279, rz=-0.000461, shoulder=lefty, elbow=epositive, wrist=wpositive, fatherId=frmaster[1]}
  [552] = {x=-62.950739, y=-2.831421, z=112.320225, rx=179.999902, ry=-5.779447, rz=0.000511, shoulder=lefty, elbow=epositive, wrist=wpositive, fatherId=frmaster[1]}
  [553] = {x=-62.948805, y=-2.831104, z=102.322171, rx=179.999806, ry=-5.778638, rz=0.000974, shoulder=lefty, elbow=epositive, wrist=wpositive, fatherId=frmaster[1]}
  [554] = {x=-59.392635, y=-2.917312, z=104.605387, rx=179.999648, ry=-7.917177, rz=0.000694, shoulder=lefty, elbow=epositive, wrist=wpositive, fatherId=frmaster[1]}
  [555] = {x=-54.977712, y=-3.002197, z=107.153689, rx=-179.999857, ry=-10.471642, rz=-0.000229, shoulder=lefty, elbow=epositive, wrist=wpositive, fatherId=frmaster[1]}
  [556] = {x=-51.112634, y=-3.073917, z=109.115526, rx=-179.999596, ry=-12.593219, rz=-0.000606, shoulder=lefty, elbow=epositive, wrist=wpositive, fatherId=frmaster[1]}
  [557] = {x=-47.122152, y=-3.139696, z=110.968551, rx=-179.999977, ry=-14.747784, rz=-0.000261, shoulder=lefty, elbow=epositive, wrist=wpositive, fatherId=frmaster[1]}
  [558] = {x=-43.085732, y=-3.206892, z=112.647942, rx=-179.999672, ry=-16.88917, rz=0.000135, shoulder=lefty, elbow=epositive, wrist=wpositive, fatherId=frmaster[1]}
  [559] = {x=-39.003251, y=-3.272146, z=114.17975, rx=-179.999681, ry=-19.023922, rz=-0.000154, shoulder=lefty, elbow=epositive, wrist=wpositive, fatherId=frmaster[1]}
  [560] = {x=-35.225354, y=-3.365608, z=115.441359, rx=-179.999715, ry=-20.972966, rz=-0.000202, shoulder=lefty, elbow=epositive, wrist=wpositive, fatherId=frmaster[1]}
  [561] = {x=-31.372851, y=-3.455581, z=116.590195, rx=179.999812, ry=-22.941009, rz=0.000012, shoulder=lefty, elbow=epositive, wrist=wpositive, fatherId=frmaster[1]}
  [562] = {x=-27.439752, y=-3.545534, z=117.607898, rx=179.999933, ry=-24.92892, rz=-0.000011, shoulder=lefty, elbow=epositive, wrist=wpositive, fatherId=frmaster[1]}
  [563] = {x=-23.424324, y=-3.641627, z=118.502477, rx=179.999393, ry=-26.940569, rz=-0.000425, shoulder=lefty, elbow=epositive, wrist=wpositive, fatherId=frmaster[1]}
  [564] = {x=-19.772027, y=-3.750742, z=119.178462, rx=-179.999966, ry=-28.754908, rz=-0.000652, shoulder=lefty, elbow=epositive, wrist=wpositive, fatherId=frmaster[1]}
  [565] = {x=-16.024713, y=-3.85535, z=119.763267, rx=-179.999826, ry=-30.609619, rz=-0.000414, shoulder=lefty, elbow=epositive, wrist=wpositive, fatherId=frmaster[1]}
  [566] = {x=-12.170244, y=-3.966813, z=120.227225, rx=-179.999802, ry=-32.50284, rz=0.00014, shoulder=lefty, elbow=epositive, wrist=wpositive, fatherId=frmaster[1]}
  [567] = {x=-8.221299, y=-4.077638, z=120.574314, rx=179.999538, ry=-34.43874, rz=-0.000576, shoulder=lefty, elbow=epositive, wrist=wpositive, fatherId=frmaster[1]}
  [568] = {x=-2.619902, y=-4.171781, z=120.831867, rx=179.99949, ry=-37.131331, rz=-0.001232, shoulder=lefty, elbow=epositive, wrist=wpositive, fatherId=frmaster[1]}
  [569] = {x=0.625696, y=-4.19881, z=120.854669, rx=-179.999382, ry=-38.681586, rz=0.000272, shoulder=lefty, elbow=epositive, wrist=wpositive, fatherId=frmaster[1]}
  [570] = {x=6.74505, y=-4.263301, z=120.667544, rx=179.999605, ry=-41.609141, rz=0.000198, shoulder=lefty, elbow=epositive, wrist=wpositive, fatherId=frmaster[1]}
  [571] = {x=12.282991, y=-4.321833, z=120.22316, rx=179.999927, ry=-44.266878, rz=0.000005, shoulder=lefty, elbow=epositive, wrist=wpositive, fatherId=frmaster[1]}
  [572] = {x=17.183154, y=-4.381587, z=119.617931, rx=-179.999602, ry=-46.632554, rz=0.000055, shoulder=lefty, elbow=epositive, wrist=wpositive, fatherId=frmaster[1]}
  [573] = {x=21.437621, y=-4.447851, z=118.918382, rx=-179.999791, ry=-48.698544, rz=-0.000418, shoulder=lefty, elbow=epositive, wrist=wpositive, fatherId=frmaster[1]}
  [574] = {x=25.058927, y=-4.51065, z=118.196775, rx=179.999364, ry=-50.471579, rz=-0.000889, shoulder=lefty, elbow=epositive, wrist=wpositive, fatherId=frmaster[1]}
  [575] = {x=28.077555, y=-4.568242, z=117.506921, rx=-179.999737, ry=-51.963472, rz=0.000334, shoulder=lefty, elbow=epositive, wrist=wpositive, fatherId=frmaster[1]}
  [576] = {x=32.196295, y=-4.704318, z=116.429731, rx=179.999097, ry=-54.025943, rz=-0.000441, shoulder=lefty, elbow=epositive, wrist=wpositive, fatherId=frmaster[1]}
  [577] = {x=34.713857, y=-5.096181, z=115.619962, rx=-179.999274, ry=-55.403761, rz=0.000748, shoulder=lefty, elbow=epositive, wrist=wpositive, fatherId=frmaster[1]}
  [578] = {x=38.128278, y=-5.36519, z=114.490617, rx=-179.999478, ry=-57.187533, rz=0.000789, shoulder=lefty, elbow=epositive, wrist=wpositive, fatherId=frmaster[1]}
  [579] = {x=43.907048, y=-5.500534, z=112.366135, rx=179.999467, ry=-60.146554, rz=-0.001285, shoulder=lefty, elbow=epositive, wrist=wpositive, fatherId=frmaster[1]}
  [580] = {x=49.396483, y=-5.636896, z=110.028606, rx=-179.999982, ry=-63.019037, rz=-0.000193, shoulder=lefty, elbow=epositive, wrist=wpositive, fatherId=frmaster[1]}
  [581] = {x=54.602429, y=-5.769603, z=107.499828, rx=-179.999459, ry=-65.805379, rz=0.000237, shoulder=lefty, elbow=epositive, wrist=wpositive, fatherId=frmaster[1]}
  [582] = {x=59.531852, y=-5.906344, z=104.800304, rx=-179.999548, ry=-68.512721, rz=0.00041, shoulder=lefty, elbow=epositive, wrist=wpositive, fatherId=frmaster[1]}
  [583] = {x=64.207082, y=-6.042768, z=101.954543, rx=179.998043, ry=-71.148488, rz=-0.002531, shoulder=lefty, elbow=epositive, wrist=wpositive, fatherId=frmaster[1]}
  [584] = {x=68.638271, y=-6.177985, z=98.971825, rx=179.998397, ry=-73.724282, rz=-0.000879, shoulder=lefty, elbow=epositive, wrist=wpositive, fatherId=frmaster[1]}
  [585] = {x=72.711221, y=-6.310383, z=95.957311, rx=-179.999359, ry=-76.167773, rz=0.001114, shoulder=lefty, elbow=epositive, wrist=wpositive, fatherId=frmaster[1]}
  [586] = {x=76.690253, y=-6.447978, z=92.744539, rx=-179.999215, ry=-78.630237, rz=0.001211, shoulder=lefty, elbow=epositive, wrist=wpositive, fatherId=frmaster[1]}
  [587] = {x=79.76531, y=-6.590526, z=90.046224, rx=179.99652, ry=-80.609063, rz=-0.002905, shoulder=lefty, elbow=epositive, wrist=wpositive, fatherId=frmaster[1]}
  [588] = {x=81.292794, y=-6.725135, z=88.59474, rx=179.998632, ry=-81.637991, rz=-0.001566, shoulder=lefty, elbow=epositive, wrist=wpositive, fatherId=frmaster[1]}
  [589] = {x=84.157063, y=-7.00207, z=85.724822, rx=179.994196, ry=-83.625908, rz=-0.005297, shoulder=lefty, elbow=epositive, wrist=wpositive, fatherId=frmaster[1]}
  [590] = {x=86.778949, y=-7.275345, z=82.906184, rx=179.996751, ry=-85.516095, rz=-0.002927, shoulder=lefty, elbow=epositive, wrist=wpositive, fatherId=frmaster[1]}
  [591] = {x=89.186207, y=-7.549443, z=80.12928, rx=179.995313, ry=-87.321134, rz=-0.004564, shoulder=lefty, elbow=epositive, wrist=wpositive, fatherId=frmaster[1]}
  [592] = {x=91.394473, y=-7.82889, z=77.420107, rx=179.943452, ry=-89.043955, rz=-0.056967, shoulder=lefty, elbow=epositive, wrist=wpositive, fatherId=frmaster[1]}
  [593] = {x=93.406759, y=-8.097459, z=74.778084, rx=-0.045088, ry=-89.319041, rz=179.955183, shoulder=lefty, elbow=epositive, wrist=wpositive, fatherId=frmaster[1]}
  [594] = {x=95.237125, y=-8.371727, z=72.224832, rx=-0.019963, ry=-87.765865, rz=179.980735, shoulder=lefty, elbow=epositive, wrist=wpositive, fatherId=frmaster[1]}
  [595] = {x=98.501619, y=-8.92147, z=67.236292, rx=0.004349, ry=-84.820122, rz=-179.995722, shoulder=lefty, elbow=epositive, wrist=wpositive, fatherId=frmaster[1]}
  [596] = {x=101.172292, y=-9.462736, z=62.615108, rx=-0.003149, ry=-82.167319, rz=179.996319, shoulder=lefty, elbow=epositive, wrist=wpositive, fatherId=frmaster[1]}
  [597] = {x=103.354264, y=-10.011064, z=58.377762, rx=0.001667, ry=-79.792745, rz=-179.998472, shoulder=lefty, elbow=epositive, wrist=wpositive, fatherId=frmaster[1]}
  [598] = {x=105.11552, y=-10.55484, z=54.516735, rx=-0.000658, ry=-77.673891, rz=179.998869, shoulder=lefty, elbow=epositive, wrist=wpositive, fatherId=frmaster[1]}
  [599] = {x=103.838916, y=-12.720111, z=54.353603, rx=0.001933, ry=-77.581832, rz=-179.998054, shoulder=lefty, elbow=epositive, wrist=wpositive, fatherId=frmaster[1]}
  [600] = {x=102.438989, y=-14.858388, z=54.355475, rx=0.000543, ry=-77.581969, rz=-179.999153, shoulder=lefty, elbow=epositive, wrist=wpositive, fatherId=frmaster[1]}
  [601] = {x=101.008134, y=-16.972391, z=54.350105, rx=-0.002926, ry=-77.582005, rz=179.996693, shoulder=lefty, elbow=epositive, wrist=wpositive, fatherId=frmaster[1]}
  [602] = {x=99.548937, y=-19.06947, z=54.350705, rx=-0.001699, ry=-77.582192, rz=179.998525, shoulder=lefty, elbow=epositive, wrist=wpositive, fatherId=frmaster[1]}
  [603] = {x=98.054006, y=-21.14454, z=54.354844, rx=-0.002018, ry=-77.581524, rz=179.997977, shoulder=lefty, elbow=epositive, wrist=wpositive, fatherId=frmaster[1]}
  [604] = {x=96.534028, y=-23.197602, z=54.354616, rx=0.00199, ry=-77.581438, rz=-179.998328, shoulder=lefty, elbow=epositive, wrist=wpositive, fatherId=frmaster[1]}
  [605] = {x=97.868761, y=-22.257232, z=54.355898, rx=0.002513, ry=-77.581721, rz=-179.996929, shoulder=lefty, elbow=epositive, wrist=wpositive, fatherId=frmaster[1]}
  [606] = {x=99.204107, y=-21.313765, z=54.356144, rx=-0.000838, ry=-77.581259, rz=179.99992, shoulder=lefty, elbow=epositive, wrist=wpositive, fatherId=frmaster[1]}
  [607] = {x=100.50959, y=-20.331581, z=54.349013, rx=-0.001117, ry=-77.582816, rz=179.99914, shoulder=lefty, elbow=epositive, wrist=wpositive, fatherId=frmaster[1]}
  [608] = {x=101.815349, y=-19.348291, z=54.349067, rx=-0.001727, ry=-77.582525, rz=179.997693, shoulder=lefty, elbow=epositive, wrist=wpositive, fatherId=frmaster[1]}
  [609] = {x=103.069361, y=-18.311831, z=54.354466, rx=0.003955, ry=-77.58189, rz=-179.99594, shoulder=lefty, elbow=epositive, wrist=wpositive, fatherId=frmaster[1]}
  [610] = {x=104.266654, y=-17.20492, z=54.353712, rx=-0.00189, ry=-77.582315, rz=179.9987, shoulder=lefty, elbow=epositive, wrist=wpositive, fatherId=frmaster[1]}
  [611] = {x=104.190532, y=-16.029161, z=56.599085, rx=0.002104, ry=-78.811835, rz=-179.997519, shoulder=lefty, elbow=epositive, wrist=wpositive, fatherId=frmaster[1]}
  [612] = {x=102.7239, y=-15.709302, z=59.65471, rx=0.001303, ry=-80.506995, rz=-179.999089, shoulder=lefty, elbow=epositive, wrist=wpositive, fatherId=frmaster[1]}
  [613] = {x=101.003388, y=-15.394111, z=62.932079, rx=0.004031, ry=-82.348046, rz=-179.995883, shoulder=lefty, elbow=epositive, wrist=wpositive, fatherId=frmaster[1]}
  [614] = {x=99.243261, y=-15.049962, z=66.00079, rx=-0.002109, ry=-84.107191, rz=179.997523, shoulder=lefty, elbow=epositive, wrist=wpositive, fatherId=frmaster[1]}
  [615] = {x=97.232339, y=-14.717157, z=69.250598, rx=0.004793, ry=-85.99494, rz=-179.995186, shoulder=lefty, elbow=epositive, wrist=wpositive, fatherId=frmaster[1]}
  [616] = {x=95.347548, y=-14.355907, z=72.062961, rx=-0.011463, ry=-87.673062, rz=179.988472, shoulder=lefty, elbow=epositive, wrist=wpositive, fatherId=frmaster[1]}
  [617] = {x=93.247331, y=-13.99959, z=74.994562, rx=-0.0404, ry=-89.451103, rz=179.959838, shoulder=lefty, elbow=epositive, wrist=wpositive, fatherId=frmaster[1]}
  [618] = {x=89.810335, y=-13.239854, z=79.376577, rx=179.997642, ry=-87.80259, rz=-0.003132, shoulder=lefty, elbow=epositive, wrist=wpositive, fatherId=frmaster[1]}
  [619] = {x=88.256708, y=-12.656609, z=81.22389, rx=179.997971, ry=-86.613703, rz=-0.002424, shoulder=lefty, elbow=epositive, wrist=wpositive, fatherId=frmaster[1]}
  [620] = {x=88.527883, y=-11.633174, z=80.913929, rx=179.987496, ry=-86.82157, rz=-0.012672, shoulder=lefty, elbow=epositive, wrist=wpositive, fatherId=frmaster[1]}
  [621] = {x=91.40138, y=-10.883918, z=77.411685, rx=179.970092, ry=-89.048093, rz=-0.029739, shoulder=lefty, elbow=epositive, wrist=wpositive, fatherId=frmaster[1]}
  [622] = {x=94.52657, y=-10.358568, z=73.233909, rx=0.001477, ry=-88.37834, rz=-179.999206, shoulder=lefty, elbow=epositive, wrist=wpositive, fatherId=frmaster[1]}
  [623] = {x=97.830801, y=-9.871919, z=68.309417, rx=0.002049, ry=-85.446203, rz=-179.998129, shoulder=lefty, elbow=epositive, wrist=wpositive, fatherId=frmaster[1]}
  [624] = {x=99.476008, y=-9.642282, z=65.615065, rx=-0.004839, ry=-83.88021, rz=179.994848, shoulder=lefty, elbow=epositive, wrist=wpositive, fatherId=frmaster[1]}
  [625] = {x=100.943329, y=-9.411664, z=63.033007, rx=-0.003901, ry=-82.40857, rz=179.995575, shoulder=lefty, elbow=epositive, wrist=wpositive, fatherId=frmaster[1]}
  [626] = {x=103.64712, y=-8.986784, z=57.761453, rx=-0.003458, ry=-79.451137, rz=179.996862, shoulder=lefty, elbow=epositive, wrist=wpositive, fatherId=frmaster[1]}
  [627] = {x=104.253325, y=-7.928501, z=54.353207, rx=0.001066, ry=-77.581955, rz=-179.998751, shoulder=lefty, elbow=epositive, wrist=wpositive, fatherId=frmaster[1]}
  [628] = {x=102.289316, y=-6.505284, z=54.354094, rx=0.002721, ry=-77.582083, rz=-179.997039, shoulder=lefty, elbow=epositive, wrist=wpositive, fatherId=frmaster[1]}
  [629] = {x=100.275033, y=-5.147438, z=54.353397, rx=0.001126, ry=-77.582173, rz=-179.998485, shoulder=lefty, elbow=epositive, wrist=wpositive, fatherId=frmaster[1]}
  [630] = {x=98.952, y=-4.206239, z=54.348687, rx=-0.000336, ry=-77.582486, rz=179.999309, shoulder=lefty, elbow=epositive, wrist=wpositive, fatherId=frmaster[1]}
  [631] = {x=97.685935, y=-3.198636, z=54.352063, rx=-0.001451, ry=-77.58197, rz=179.998382, shoulder=lefty, elbow=epositive, wrist=wpositive, fatherId=frmaster[1]}
  [632] = {x=97.103843, y=-2.658134, z=54.355974, rx=0.00071, ry=-77.581483, rz=-179.998739, shoulder=lefty, elbow=epositive, wrist=wpositive, fatherId=frmaster[1]}
  [633] = {x=96.398883, y=-1.703119, z=54.354736, rx=-0.003446, ry=-77.581494, rz=179.996512, shoulder=lefty, elbow=epositive, wrist=wpositive, fatherId=frmaster[1]}
  [634] = {x=96.195277, y=-1.152172, z=54.35215, rx=-0.000728, ry=-77.582218, rz=179.999193, shoulder=lefty, elbow=epositive, wrist=wpositive, fatherId=frmaster[1]}
  [635] = {x=96.189014, y=-0.573216, z=54.355644, rx=-0.001771, ry=-77.581601, rz=179.998859, shoulder=lefty, elbow=epositive, wrist=wpositive, fatherId=frmaster[1]}
  [636] = {x=96.298853, y=-0.20119, z=54.353906, rx=0.003345, ry=-77.581906, rz=-179.997266, shoulder=lefty, elbow=epositive, wrist=wpositive, fatherId=frmaster[1]}
  [637] = {x=96.684682, y=0.430738, z=54.356497, rx=-0.000857, ry=-77.581193, rz=179.999119, shoulder=lefty, elbow=epositive, wrist=wpositive, fatherId=frmaster[1]}
  [638] = {x=97.566262, y=1.280654, z=54.353314, rx=-0.002039, ry=-77.581938, rz=179.998064, shoulder=lefty, elbow=epositive, wrist=wpositive, fatherId=frmaster[1]}
  [639] = {x=98.391656, y=1.875075, z=54.353135, rx=0.001583, ry=-77.582027, rz=-179.99895, shoulder=lefty, elbow=epositive, wrist=wpositive, fatherId=frmaster[1]}
  [640] = {x=99.683726, y=2.677599, z=54.354594, rx=0.000743, ry=-77.581612, rz=-179.998832, shoulder=lefty, elbow=epositive, wrist=wpositive, fatherId=frmaster[1]}
  [641] = {x=100.978627, y=3.484732, z=54.350033, rx=-0.002081, ry=-77.582152, rz=179.997929, shoulder=lefty, elbow=epositive, wrist=wpositive, fatherId=frmaster[1]}
  [642] = {x=102.354329, y=4.321963, z=54.352569, rx=0.001081, ry=-77.581314, rz=-179.999455, shoulder=lefty, elbow=epositive, wrist=wpositive, fatherId=frmaster[1]}
  [643] = {x=104.306362, y=5.72215, z=54.356875, rx=-0.000168, ry=-77.58137, rz=-179.99998, shoulder=lefty, elbow=epositive, wrist=wpositive, fatherId=frmaster[1]}
  [644] = {x=103.054099, y=6.994717, z=58.98914, rx=0.002769, ry=-80.133089, rz=-179.997248, shoulder=lefty, elbow=epositive, wrist=wpositive, fatherId=frmaster[1]}
  [645] = {x=100.773879, y=7.483944, z=63.346445, rx=0.002442, ry=-82.584101, rz=-179.997196, shoulder=lefty, elbow=epositive, wrist=wpositive, fatherId=frmaster[1]}
  [646] = {x=97.946015, y=8.188977, z=68.126988, rx=-0.002555, ry=-85.340869, rz=179.997579, shoulder=lefty, elbow=epositive, wrist=wpositive, fatherId=frmaster[1]}
  [647] = {x=96.122064, y=8.94264, z=70.930985, rx=-0.005507, ry=-86.99368, rz=179.994476, shoulder=lefty, elbow=epositive, wrist=wpositive, fatherId=frmaster[1]}
  [648] = {x=95.793314, y=9.524517, z=71.41867, rx=0.001613, ry=-87.28857, rz=-179.998953, shoulder=lefty, elbow=epositive, wrist=wpositive, fatherId=frmaster[1]}
  [649] = {x=97.038054, y=10.534031, z=69.550683, rx=0.006081, ry=-86.172677, rz=-179.993924, shoulder=lefty, elbow=epositive, wrist=wpositive, fatherId=frmaster[1]}
  [650] = {x=99.762592, y=11.512517, z=65.123355, rx=0.000457, ry=-83.600115, rz=-179.999498, shoulder=lefty, elbow=epositive, wrist=wpositive, fatherId=frmaster[1]}
  [651] = {x=101.473827, y=11.990986, z=62.060819, rx=-0.000416, ry=-81.856005, rz=179.999574, shoulder=lefty, elbow=epositive, wrist=wpositive, fatherId=frmaster[1]}
  [652] = {x=102.963785, y=12.469917, z=59.177367, rx=-0.00099, ry=-80.236803, rz=179.99938, shoulder=lefty, elbow=epositive, wrist=wpositive, fatherId=frmaster[1]}
  [653] = {x=105.060152, y=13.380897, z=54.348574, rx=-0.000655, ry=-77.582344, rz=179.998916, shoulder=lefty, elbow=epositive, wrist=wpositive, fatherId=frmaster[1]}
  [654] = {x=104.134686, y=14.717449, z=54.350609, rx=0.000885, ry=-77.582224, rz=-179.999446, shoulder=lefty, elbow=epositive, wrist=wpositive, fatherId=frmaster[1]}
  [655] = {x=102.603083, y=16.610601, z=54.354991, rx=-0.001344, ry=-77.58178, rz=179.998266, shoulder=lefty, elbow=epositive, wrist=wpositive, fatherId=frmaster[1]}
  [656] = {x=100.970912, y=18.421275, z=54.354642, rx=0.002338, ry=-77.582009, rz=-179.997296, shoulder=lefty, elbow=epositive, wrist=wpositive, fatherId=frmaster[1]}
  [657] = {x=99.86499, y=19.617705, z=54.351951, rx=0.002184, ry=-77.581861, rz=-179.998442, shoulder=lefty, elbow=epositive, wrist=wpositive, fatherId=frmaster[1]}
  [658] = {x=98.756686, y=20.814021, z=54.355158, rx=0.001899, ry=-77.581472, rz=-179.99798, shoulder=lefty, elbow=epositive, wrist=wpositive, fatherId=frmaster[1]}
  [659] = {x=97.643595, y=22.00981, z=54.353004, rx=-0.002253, ry=-77.581946, rz=179.998084, shoulder=lefty, elbow=epositive, wrist=wpositive, fatherId=frmaster[1]}
  [660] = {x=96.529068, y=23.197406, z=54.35321, rx=-0.002023, ry=-77.582158, rz=179.99835, shoulder=lefty, elbow=epositive, wrist=wpositive, fatherId=frmaster[1]}
  [661] = {x=98.058228, y=21.145694, z=54.351986, rx=-0.00148, ry=-77.582094, rz=179.998195, shoulder=lefty, elbow=epositive, wrist=wpositive, fatherId=frmaster[1]}
  [662] = {x=99.551075, y=19.06641, z=54.354891, rx=0.001836, ry=-77.581772, rz=-179.997755, shoulder=lefty, elbow=epositive, wrist=wpositive, fatherId=frmaster[1]}
  [663] = {x=101.011695, y=16.971786, z=54.356201, rx=-0.00253, ry=-77.581304, rz=179.998276, shoulder=lefty, elbow=epositive, wrist=wpositive, fatherId=frmaster[1]}
  [664] = {x=102.444384, y=14.851817, z=54.354322, rx=0.001627, ry=-77.582042, rz=-179.998014, shoulder=lefty, elbow=epositive, wrist=wpositive, fatherId=frmaster[1]}
  [665] = {x=103.8426, y=12.711063, z=54.354862, rx=0.002046, ry=-77.58167, rz=-179.997895, shoulder=lefty, elbow=epositive, wrist=wpositive, fatherId=frmaster[1]}
  [666] = {x=105.090753, y=10.547702, z=54.578679, rx=0.002028, ry=-77.703349, rz=-179.998091, shoulder=lefty, elbow=epositive, wrist=wpositive, fatherId=frmaster[1]}
  [667] = {x=103.316892, y=10.002592, z=58.451556, rx=-0.00052, ry=-79.836819, rz=179.999184, shoulder=lefty, elbow=epositive, wrist=wpositive, fatherId=frmaster[1]}
  [668] = {x=101.123988, y=9.454827, z=62.711584, rx=0.004046, ry=-82.222765, rz=-179.996051, shoulder=lefty, elbow=epositive, wrist=wpositive, fatherId=frmaster[1]}
  [669] = {x=98.433413, y=8.908507, z=67.347732, rx=0.00078, ry=-84.884833, rz=-179.999428, shoulder=lefty, elbow=epositive, wrist=wpositive, fatherId=frmaster[1]}
  [670] = {x=95.159578, y=8.363697, z=72.33948, rx=0.005676, ry=-87.836745, rz=-179.994606, shoulder=lefty, elbow=epositive, wrist=wpositive, fatherId=frmaster[1]}
  [671] = {x=93.323195, y=8.088357, z=74.892364, rx=0.0084, ry=-89.388719, rz=-179.991164, shoulder=lefty, elbow=epositive, wrist=wpositive, fatherId=frmaster[1]}
  [672] = {x=91.308188, y=7.81339, z=77.53028, rx=-179.992515, ry=-88.975674, rz=0.006962, shoulder=lefty, elbow=epositive, wrist=wpositive, fatherId=frmaster[1]}
  [673] = {x=89.095211, y=7.538581, z=80.235864, rx=-179.987676, ry=-87.253868, rz=0.012538, shoulder=lefty, elbow=epositive, wrist=wpositive, fatherId=frmaster[1]}
  [674] = {x=86.686101, y=7.262227, z=83.00623, rx=-179.998713, ry=-85.448628, rz=0.000833, shoulder=lefty, elbow=epositive, wrist=wpositive, fatherId=frmaster[1]}
  [675] = {x=84.061675, y=6.987643, z=85.817003, rx=-179.998309, ry=-83.559913, rz=0.001738, shoulder=lefty, elbow=epositive, wrist=wpositive, fatherId=frmaster[1]}
  [676] = {x=81.198206, y=6.711042, z=88.683127, rx=179.997681, ry=-81.573854, rz=-0.002723, shoulder=lefty, elbow=epositive, wrist=wpositive, fatherId=frmaster[1]}
  [677] = {x=79.668629, y=6.573204, z=90.132289, rx=179.998766, ry=-80.544761, rz=-0.001268, shoulder=lefty, elbow=epositive, wrist=wpositive, fatherId=frmaster[1]}
  [678] = {x=76.462994, y=6.439004, z=92.928816, rx=-179.999068, ry=-78.487346, rz=0.00037, shoulder=lefty, elbow=epositive, wrist=wpositive, fatherId=frmaster[1]}
  [679] = {x=72.501248, y=6.297825, z=96.122515, rx=179.998457, ry=-76.037694, rz=-0.00189, shoulder=lefty, elbow=epositive, wrist=wpositive, fatherId=frmaster[1]}
  [680] = {x=68.430611, y=6.160737, z=99.118699, rx=179.998641, ry=-73.60261, rz=-0.00109, shoulder=lefty, elbow=epositive, wrist=wpositive, fatherId=frmaster[1]}
  [681] = {x=64.026745, y=6.026268, z=102.070371, rx=179.999855, ry=-71.045137, rz=-0.000403, shoulder=lefty, elbow=epositive, wrist=wpositive, fatherId=frmaster[1]}
  [682] = {x=59.385098, y=5.89071, z=104.885761, rx=179.998845, ry=-68.428276, rz=-0.001955, shoulder=lefty, elbow=epositive, wrist=wpositive, fatherId=frmaster[1]}
  [683] = {x=54.492378, y=5.755417, z=107.551317, rx=179.999315, ry=-65.743901, rz=-0.001118, shoulder=lefty, elbow=epositive, wrist=wpositive, fatherId=frmaster[1]}
  [684] = {x=49.327962, y=5.625171, z=110.062084, rx=-179.999722, ry=-62.984616, rz=-0.000131, shoulder=lefty, elbow=epositive, wrist=wpositive, fatherId=frmaster[1]}
  [685] = {x=43.898282, y=5.48751, z=112.368158, rx=179.999978, ry=-60.141383, rz=-0.00038, shoulder=lefty, elbow=epositive, wrist=wpositive, fatherId=frmaster[1]}
  [686] = {x=38.18975, y=5.34917, z=114.466811, rx=179.998744, ry=-57.216429, rz=-0.001681, shoulder=lefty, elbow=epositive, wrist=wpositive, fatherId=frmaster[1]}
  [687] = {x=34.621987, y=4.823039, z=115.700057, rx=-179.999286, ry=-55.267079, rz=0.000952, shoulder=lefty, elbow=epositive, wrist=wpositive, fatherId=frmaster[1]}
  [688] = {x=32.145289, y=4.688988, z=116.443192, rx=179.998591, ry=-53.999011, rz=-0.001506, shoulder=lefty, elbow=epositive, wrist=wpositive, fatherId=frmaster[1]}
  [689] = {x=27.941453, y=4.558477, z=117.539041, rx=179.999138, ry=-51.89525, rz=-0.001937, shoulder=lefty, elbow=epositive, wrist=wpositive, fatherId=frmaster[1]}
  [690] = {x=24.921268, y=4.496263, z=118.233929, rx=179.999411, ry=-50.405439, rz=-0.000059, shoulder=lefty, elbow=epositive, wrist=wpositive, fatherId=frmaster[1]}
  [691] = {x=21.319468, y=4.433456, z=118.940164, rx=179.999068, ry=-48.640684, rz=-0.00157, shoulder=lefty, elbow=epositive, wrist=wpositive, fatherId=frmaster[1]}
  [692] = {x=17.105294, y=4.37275, z=119.625706, rx=-179.999902, ry=-46.592221, rz=-0.000376, shoulder=lefty, elbow=epositive, wrist=wpositive, fatherId=frmaster[1]}
  [693] = {x=12.264052, y=4.311554, z=120.231894, rx=179.999801, ry=-44.25748, rz=-0.00034, shoulder=lefty, elbow=epositive, wrist=wpositive, fatherId=frmaster[1]}
  [694] = {x=6.814915, y=4.251282, z=120.666729, rx=-179.999794, ry=-41.642549, rz=0.000561, shoulder=lefty, elbow=epositive, wrist=wpositive, fatherId=frmaster[1]}
  [695] = {x=0.816219, y=4.186945, z=120.850438, rx=179.999642, ry=-38.772931, rz=-0.000688, shoulder=lefty, elbow=epositive, wrist=wpositive, fatherId=frmaster[1]}
  [696] = {x=-2.359525, y=4.154634, z=120.837723, rx=179.999195, ry=-37.25664, rz=0.00012, shoulder=lefty, elbow=epositive, wrist=wpositive, fatherId=frmaster[1]}
  [697] = {x=-8.110342, y=4.065925, z=120.579428, rx=-179.999818, ry=-34.491809, rz=0.000245, shoulder=lefty, elbow=epositive, wrist=wpositive, fatherId=frmaster[1]}
  [698] = {x=-12.016553, y=3.95663, z=120.242007, rx=179.999955, ry=-32.578698, rz=-0.000057, shoulder=lefty, elbow=epositive, wrist=wpositive, fatherId=frmaster[1]}
  [699] = {x=-15.824238, y=3.844674, z=119.784342, rx=-179.999843, ry=-30.705837, rz=0.000022, shoulder=lefty, elbow=epositive, wrist=wpositive, fatherId=frmaster[1]}
  [700] = {x=-19.535632, y=3.735207, z=119.223589, rx=-179.999922, ry=-28.872751, rz=-0.000136, shoulder=lefty, elbow=epositive, wrist=wpositive, fatherId=frmaster[1]}
  [701] = {x=-23.146692, y=3.626679, z=118.554197, rx=179.999907, ry=-27.076952, rz=-0.000099, shoulder=lefty, elbow=epositive, wrist=wpositive, fatherId=frmaster[1]}
  [702] = {x=-27.144358, y=3.539542, z=117.677895, rx=-179.999478, ry=-25.075797, rz=0.00002, shoulder=lefty, elbow=epositive, wrist=wpositive, fatherId=frmaster[1]}
  [703] = {x=-31.063469, y=3.449357, z=116.667617, rx=-179.999264, ry=-23.096041, rz=-0.000293, shoulder=lefty, elbow=epositive, wrist=wpositive, fatherId=frmaster[1]}
  [704] = {x=-34.900159, y=3.355192, z=115.539023, rx=-179.999653, ry=-21.136993, rz=-0.000645, shoulder=lefty, elbow=epositive, wrist=wpositive, fatherId=frmaster[1]}
  [705] = {x=-38.669291, y=3.267622, z=114.297328, rx=179.999639, ry=-19.197361, rz=0.00007, shoulder=lefty, elbow=epositive, wrist=wpositive, fatherId=frmaster[1]}
  [706] = {x=-42.772471, y=3.202028, z=112.773509, rx=-179.999697, ry=-17.052761, rz=0.000153, shoulder=lefty, elbow=epositive, wrist=wpositive, fatherId=frmaster[1]}
  [707] = {x=-46.831086, y=3.134799, z=111.092455, rx=179.999571, ry=-14.902493, rz=0.000045, shoulder=lefty, elbow=epositive, wrist=wpositive, fatherId=frmaster[1]}
  [708] = {x=-50.844636, y=3.06516, z=109.251815, rx=179.999993, ry=-12.740784, rz=0.000247, shoulder=lefty, elbow=epositive, wrist=wpositive, fatherId=frmaster[1]}
  [709] = {x=-54.814615, y=2.997805, z=107.240668, rx=-179.999527, ry=-10.561904, rz=-0.000413, shoulder=lefty, elbow=epositive, wrist=wpositive, fatherId=frmaster[1]}
  [710] = {x=-59.327534, y=2.912938, z=104.641902, rx=-179.999886, ry=-7.953301, rz=-0.000394, shoulder=lefty, elbow=epositive, wrist=wpositive, fatherId=frmaster[1]}
  [711] = {x=-62.947412, y=2.832964, z=102.322113, rx=179.999805, ry=-5.779294, rz=-0.000037, shoulder=lefty, elbow=epositive, wrist=wpositive, fatherId=frmaster[1]}
  [712] = {x=-62.947085, y=2.832936, z=112.317767, rx=179.999789, ry=-5.77901, rz=0.00026, shoulder=lefty, elbow=epositive, wrist=wpositive, fatherId=frmaster[1]}
pointRx pdemo2[1183]
  [0] = {x=-65.422998, y=-3.678422, z=122.358447, rx=-179.999982, ry=-2.000361, rz=-0.000689, shoulder=lefty, elbow=epositive, wrist=wpositive, fatherId=frmaster[2]}
  [1] = {x=-65.924201, y=-3.67615, z=107.996596, rx=-179.999579, ry=-1.999732, rz=0.000043, shoulder=lefty, elbow=epositive, wrist=wpositive, fatherId=frmaster[2]}
  [2] = {x=-65.92118, y=-3.67617, z=97.99056, rx=-179.999383, ry=-1.999677, rz=-0.00073, shoulder=lefty, elbow=epositive, wrist=wpositive, fatherId=frmaster[2]}
  [3] = {x=-65.954336, y=-2.699632, z=97.990625, rx=-179.999642, ry=-1.999793, rz=-0.000468, shoulder=lefty, elbow=epositive, wrist=wpositive, fatherId=frmaster[2]}
  [4] = {x=-65.987547, y=-1.724212, z=97.999229, rx=179.999104, ry=-1.99981, rz=-0.000194, shoulder=lefty, elbow=epositive, wrist=wpositive, fatherId=frmaster[2]}
  [5] = {x=-66.012678, y=-0.745327, z=97.993866, rx=179.999815, ry=-2.000016, rz=-0.000882, shoulder=lefty, elbow=epositive, wrist=wpositive, fatherId=frmaster[2]}
  [6] = {x=-66.046524, y=0.231131, z=97.99712, rx=179.999557, ry=-2.000124, rz=-0.000557, shoulder=lefty, elbow=epositive, wrist=wpositive, fatherId=frmaster[2]}
  [7] = {x=-66.080858, y=1.209717, z=97.995258, rx=-179.999705, ry=-2.000327, rz=-0.000202, shoulder=lefty, elbow=epositive, wrist=wpositive, fatherId=frmaster[2]}
  [8] = {x=-66.106558, y=2.186892, z=97.993156, rx=-179.999987, ry=-2.000418, rz=-0.000861, shoulder=lefty, elbow=epositive, wrist=wpositive, fatherId=frmaster[2]}
  [9] = {x=-66.140173, y=3.164984, z=97.994681, rx=179.999857, ry=-1.999602, rz=-0.000082, shoulder=lefty, elbow=epositive, wrist=wpositive, fatherId=frmaster[2]}
  [10] = {x=-66.166415, y=4.142612, z=97.996014, rx=179.999576, ry=-1.99969, rz=-0.000696, shoulder=lefty, elbow=epositive, wrist=wpositive, fatherId=frmaster[2]}
  [11] = {x=-66.201711, y=5.120975, z=97.992369, rx=-179.999683, ry=-1.999875, rz=-0.000279, shoulder=lefty, elbow=epositive, wrist=wpositive, fatherId=frmaster[2]}
  [12] = {x=-66.228469, y=6.098798, z=97.997142, rx=-179.999963, ry=-1.99996, rz=-0.00085, shoulder=lefty, elbow=epositive, wrist=wpositive, fatherId=frmaster[2]}
  [13] = {x=-66.264103, y=7.076026, z=97.996947, rx=179.999784, ry=-2.000032, rz=0.000575, shoulder=lefty, elbow=epositive, wrist=wpositive, fatherId=frmaster[2]}
  [14] = {x=-66.291297, y=8.05263, z=97.996566, rx=179.999505, ry=-2.000103, rz=0.000021, shoulder=lefty, elbow=epositive, wrist=wpositive, fatherId=frmaster[2]}
  [15] = {x=-66.327455, y=9.02974, z=97.991272, rx=-179.999751, ry=-2.000271, rz=0.000497, shoulder=lefty, elbow=epositive, wrist=wpositive, fatherId=frmaster[2]}
  [16] = {x=-66.355116, y=10.006033, z=97.994372, rx=179.999971, ry=-2.00034, rz=-0.000014, shoulder=lefty, elbow=epositive, wrist=wpositive, fatherId=frmaster[2]}
  [17] = {x=-66.382328, y=10.986271, z=97.996113, rx=179.999794, ry=-1.999499, rz=-0.000095, shoulder=lefty, elbow=epositive, wrist=wpositive, fatherId=frmaster[2]}
  [18] = {x=-66.419223, y=11.963259, z=97.989364, rx=-179.999461, ry=-1.999655, rz=0.000422, shoulder=lefty, elbow=epositive, wrist=wpositive, fatherId=frmaster[2]}
  [19] = {x=-66.447574, y=12.939182, z=97.999477, rx=179.999268, ry=-1.999613, rz=-0.000056, shoulder=lefty, elbow=epositive, wrist=wpositive, fatherId=frmaster[2]}
  [20] = {x=-66.476458, y=13.916554, z=97.996163, rx=179.999988, ry=-1.999768, rz=0.000505, shoulder=lefty, elbow=epositive, wrist=wpositive, fatherId=frmaster[2]}
  [21] = {x=-66.505576, y=14.894006, z=97.996411, rx=179.999713, ry=-1.999811, rz=0.000053, shoulder=lefty, elbow=epositive, wrist=wpositive, fatherId=frmaster[2]}
  [22] = {x=-66.535063, y=15.872711, z=98.000205, rx=179.999439, ry=-1.999855, rz=-0.000378, shoulder=lefty, elbow=epositive, wrist=wpositive, fatherId=frmaster[2]}
  [23] = {x=-66.573419, y=16.851584, z=97.990753, rx=-179.998819, ry=-2.000099, rz=0.000232, shoulder=lefty, elbow=epositive, wrist=wpositive, fatherId=frmaster[2]}
  [24] = {x=-66.603152, y=17.827881, z=97.998037, rx=179.999913, ry=-2.000032, rz=0.00081, shoulder=lefty, elbow=epositive, wrist=wpositive, fatherId=frmaster[2]}
  [25] = {x=-66.633393, y=18.80539, z=97.992054, rx=-179.999364, ry=-2.000165, rz=0.000428, shoulder=lefty, elbow=epositive, wrist=wpositive, fatherId=frmaster[2]}
  [26] = {x=-66.66377, y=19.782691, z=97.997995, rx=179.999369, ry=-2.000086, rz=0.000025, shoulder=lefty, elbow=epositive, wrist=wpositive, fatherId=frmaster[2]}
  [27] = {x=-66.694378, y=20.758676, z=97.99555, rx=-179.999908, ry=-2.00022, rz=-0.000314, shoulder=lefty, elbow=epositive, wrist=wpositive, fatherId=frmaster[2]}
  [28] = {x=-66.725597, y=21.738072, z=97.991832, rx=-179.999184, ry=-2.000343, rz=0.000344, shoulder=lefty, elbow=epositive, wrist=wpositive, fatherId=frmaster[2]}
  [29] = {x=-66.756606, y=22.71351, z=97.996445, rx=179.999551, ry=-2.000254, rz=-0.000019, shoulder=lefty, elbow=epositive, wrist=wpositive, fatherId=frmaster[2]}
  [30] = {x=-66.788437, y=23.693568, z=97.991458, rx=-179.999724, ry=-2.000367, rz=0.000656, shoulder=lefty, elbow=epositive, wrist=wpositive, fatherId=frmaster[2]}
  [31] = {x=-66.811974, y=24.671925, z=97.99472, rx=179.99998, ry=-2.00038, rz=-0.000655, shoulder=lefty, elbow=epositive, wrist=wpositive, fatherId=frmaster[2]}
  [32] = {x=-66.843066, y=25.650107, z=97.99324, rx=-179.999193, ry=-1.999615, rz=-0.00047, shoulder=lefty, elbow=epositive, wrist=wpositive, fatherId=frmaster[2]}
  [33] = {x=-66.875419, y=26.627703, z=97.995303, rx=-179.999461, ry=-1.999621, rz=0.00024, shoulder=lefty, elbow=epositive, wrist=wpositive, fatherId=frmaster[2]}
  [34] = {x=-66.907608, y=27.601121, z=97.99739, rx=179.999276, ry=-1.999514, rz=-0.000063, shoulder=lefty, elbow=epositive, wrist=wpositive, fatherId=frmaster[2]}
  [35] = {x=-66.940668, y=28.580148, z=97.998206, rx=-179.999997, ry=-1.999625, rz=0.000699, shoulder=lefty, elbow=epositive, wrist=wpositive, fatherId=frmaster[2]}
  [36] = {x=-66.940053, y=27.594078, z=97.994211, rx=-179.999625, ry=-1.999633, rz=0.000974, shoulder=lefty, elbow=epositive, wrist=wpositive, fatherId=frmaster[2]}
  [37] = {x=-66.939753, y=26.607486, z=97.993694, rx=179.999754, ry=-1.99953, rz=0.000236, shoulder=lefty, elbow=epositive, wrist=wpositive, fatherId=frmaster[2]}
  [38] = {x=-66.940051, y=25.622839, z=97.996685, rx=-179.999874, ry=-1.999543, rz=0.000555, shoulder=lefty, elbow=epositive, wrist=wpositive, fatherId=frmaster[2]}
  [39] = {x=-66.941826, y=24.637683, z=97.994944, rx=-179.999601, ry=-2.000426, rz=0.000407, shoulder=lefty, elbow=epositive, wrist=wpositive, fatherId=frmaster[2]}
  [40] = {x=-66.934621, y=23.653393, z=97.9966, rx=179.999752, ry=-2.000316, rz=-0.000289, shoulder=lefty, elbow=epositive, wrist=wpositive, fatherId=frmaster[2]}
  [41] = {x=-66.936175, y=22.668866, z=97.993531, rx=-179.999873, ry=-2.000308, rz=0.000046, shoulder=lefty, elbow=epositive, wrist=wpositive, fatherId=frmaster[2]}
  [42] = {x=-66.937794, y=21.681564, z=97.998786, rx=179.999507, ry=-2.000202, rz=-0.000606, shoulder=lefty, elbow=epositive, wrist=wpositive, fatherId=frmaster[2]}
  [43] = {x=-66.93997, y=20.695274, z=97.999231, rx=179.999882, ry=-2.000197, rz=-0.000226, shoulder=lefty, elbow=epositive, wrist=wpositive, fatherId=frmaster[2]}
  [44] = {x=-66.934268, y=19.709968, z=97.994759, rx=-179.999768, ry=-2.000179, rz=-0.000852, shoulder=lefty, elbow=epositive, wrist=wpositive, fatherId=frmaster[2]}
  [45] = {x=-66.9372, y=18.723343, z=97.993869, rx=179.999614, ry=-2.00005, rz=-0.000489, shoulder=lefty, elbow=epositive, wrist=wpositive, fatherId=frmaster[2]}
  [46] = {x=-66.940757, y=17.739014, z=97.996521, rx=179.999991, ry=-2.000035, rz=-0.00007, shoulder=lefty, elbow=epositive, wrist=wpositive, fatherId=frmaster[2]}
  [47] = {x=-66.936398, y=16.755794, z=97.99423, rx=-179.999657, ry=-2.000006, rz=0.000345, shoulder=lefty, elbow=epositive, wrist=wpositive, fatherId=frmaster[2]}
  [48] = {x=-66.940551, y=15.769049, z=97.991956, rx=-179.999279, ry=-1.999979, rz=0.000782, shoulder=lefty, elbow=epositive, wrist=wpositive, fatherId=frmaster[2]}
  [49] = {x=-66.936686, y=14.783465, z=97.993145, rx=-179.999921, ry=-1.99984, rz=0.000205, shoulder=lefty, elbow=epositive, wrist=wpositive, fatherId=frmaster[2]}
  [50] = {x=-66.933508, y=13.800426, z=97.989425, rx=-179.998573, ry=-1.99991, rz=-0.000306, shoulder=lefty, elbow=epositive, wrist=wpositive, fatherId=frmaster[2]}
  [51] = {x=-66.938564, y=12.811563, z=97.994172, rx=179.999817, ry=-1.999662, rz=0.000127, shoulder=lefty, elbow=epositive, wrist=wpositive, fatherId=frmaster[2]}
  [52] = {x=-66.935913, y=11.826498, z=97.993922, rx=-179.999829, ry=-1.999622, rz=-0.000376, shoulder=lefty, elbow=epositive, wrist=wpositive, fatherId=frmaster[2]}
  [53] = {x=-66.933615, y=10.841647, z=97.99723, rx=179.99953, ry=-1.999471, rz=0.000109, shoulder=lefty, elbow=epositive, wrist=wpositive, fatherId=frmaster[2]}
  [54] = {x=-66.941202, y=9.85474, z=98.000572, rx=179.999812, ry=-2.000329, rz=0.000219, shoulder=lefty, elbow=epositive, wrist=wpositive, fatherId=frmaster[2]}
  [55] = {x=-66.939546, y=8.868265, z=97.998815, rx=179.999173, ry=-2.000167, rz=-0.000277, shoulder=lefty, elbow=epositive, wrist=wpositive, fatherId=frmaster[2]}
  [56] = {x=-66.938602, y=7.884644, z=97.992053, rx=-179.999475, ry=-2.000209, rz=0.000292, shoulder=lefty, elbow=epositive, wrist=wpositive, fatherId=frmaster[2]}
  [57] = {x=-66.937649, y=6.897942, z=97.993734, rx=179.999887, ry=-2.000045, rz=-0.000161, shoulder=lefty, elbow=epositive, wrist=wpositive, fatherId=frmaster[2]}
  [58] = {x=-66.937206, y=5.912939, z=97.999001, rx=179.999249, ry=-1.99988, rz=0.000408, shoulder=lefty, elbow=epositive, wrist=wpositive, fatherId=frmaster[2]}
  [59] = {x=-66.937057, y=4.926319, z=97.995523, rx=179.999608, ry=-1.99981, rz=0.000007, shoulder=lefty, elbow=epositive, wrist=wpositive, fatherId=frmaster[2]}
  [60] = {x=-66.937429, y=3.941513, z=97.995613, rx=179.999966, ry=-1.999738, rz=0.000627, shoulder=lefty, elbow=epositive, wrist=wpositive, fatherId=frmaster[2]}
  [61] = {x=-66.938273, y=2.95741, z=97.990627, rx=-179.999674, ry=-1.999653, rz=0.000243, shoulder=lefty, elbow=epositive, wrist=wpositive, fatherId=frmaster[2]}
  [62] = {x=-66.940139, y=1.969438, z=97.999105, rx=179.999592, ry=-2.000389, rz=0.000484, shoulder=lefty, elbow=epositive, wrist=wpositive, fatherId=frmaster[2]}
  [63] = {x=-66.941755, y=0.985854, z=97.997534, rx=179.999953, ry=-2.000301, rz=0.000145, shoulder=lefty, elbow=epositive, wrist=wpositive, fatherId=frmaster[2]}
  [64] = {x=-66.934976, y=0.002086, z=97.995705, rx=-179.999712, ry=-2.00021, rz=-0.000174, shoulder=lefty, elbow=epositive, wrist=wpositive, fatherId=frmaster[2]}
  [65] = {x=-66.93708, y=-0.98407, z=97.993751, rx=-179.99935, ry=-2.000117, rz=-0.00047, shoulder=lefty, elbow=epositive, wrist=wpositive, fatherId=frmaster[2]}
  [66] = {x=-66.939242, y=-1.972654, z=98.000328, rx=179.999021, ry=-1.99982, rz=0.000211, shoulder=lefty, elbow=epositive, wrist=wpositive, fatherId=frmaster[2]}
  [67] = {x=-66.933555, y=-2.956521, z=97.992928, rx=-179.999646, ry=-1.999815, rz=-0.000035, shoulder=lefty, elbow=epositive, wrist=wpositive, fatherId=frmaster[2]}
  [68] = {x=-66.936617, y=-3.943812, z=97.994128, rx=179.999722, ry=-1.999608, rz=-0.000303, shoulder=lefty, elbow=epositive, wrist=wpositive, fatherId=frmaster[2]}
  [69] = {x=-66.941493, y=-4.927637, z=97.998977, rx=179.999989, ry=-2.000417, rz=0.000088, shoulder=lefty, elbow=epositive, wrist=wpositive, fatherId=frmaster[2]}
  [70] = {x=-66.936751, y=-5.912216, z=97.994674, rx=-179.999672, ry=-2.000298, rz=-0.000127, shoulder=lefty, elbow=epositive, wrist=wpositive, fatherId=frmaster[2]}
  [71] = {x=-66.940962, y=-6.898765, z=97.999009, rx=179.999699, ry=-2.000081, rz=0.00067, shoulder=lefty, elbow=epositive, wrist=wpositive, fatherId=frmaster[2]}
  [72] = {x=-66.936783, y=-7.884794, z=97.994173, rx=-179.999961, ry=-1.999954, rz=-0.000503, shoulder=lefty, elbow=epositive, wrist=wpositive, fatherId=frmaster[2]}
  [73] = {x=-66.933162, y=-8.868174, z=97.992923, rx=-179.99962, ry=-1.999823, rz=-0.000656, shoulder=lefty, elbow=epositive, wrist=wpositive, fatherId=frmaster[2]}
  [74] = {x=-66.938296, y=-9.856503, z=97.996454, rx=179.999752, ry=-1.999595, rz=0.000205, shoulder=lefty, elbow=epositive, wrist=wpositive, fatherId=frmaster[2]}
  [75] = {x=-66.936408, y=-10.840945, z=97.994666, rx=179.999998, ry=-2.000376, rz=-0.000288, shoulder=lefty, elbow=epositive, wrist=wpositive, fatherId=frmaster[2]}
  [76] = {x=-66.933705, y=-11.825609, z=97.992526, rx=-179.999659, ry=-2.000232, rz=-0.000375, shoulder=lefty, elbow=epositive, wrist=wpositive, fatherId=frmaster[2]}
  [77] = {x=-66.940104, y=-12.81172, z=97.999072, rx=179.999715, ry=-1.999991, rz=0.00055, shoulder=lefty, elbow=epositive, wrist=wpositive, fatherId=frmaster[2]}
  [78] = {x=-66.938061, y=-13.796784, z=97.996287, rx=-179.999941, ry=-1.999837, rz=0.000504, shoulder=lefty, elbow=epositive, wrist=wpositive, fatherId=frmaster[2]}
  [79] = {x=-66.936351, y=-14.781907, z=97.99315, rx=-179.999596, ry=-1.999677, rz=0.000478, shoulder=lefty, elbow=epositive, wrist=wpositive, fatherId=frmaster[2]}
  [80] = {x=-66.936116, y=-15.767108, z=97.989688, rx=-179.999345, ry=-2.000438, rz=0.000104, shoulder=lefty, elbow=epositive, wrist=wpositive, fatherId=frmaster[2]}
  [81] = {x=-66.934683, y=-16.755297, z=97.999844, rx=179.99901, ry=-2.000084, rz=-0.000894, shoulder=lefty, elbow=epositive, wrist=wpositive, fatherId=frmaster[2]}
  [82] = {x=-66.934156, y=-17.738788, z=97.995602, rx=-179.999647, ry=-2.00001, rz=-0.000821, shoulder=lefty, elbow=epositive, wrist=wpositive, fatherId=frmaster[2]}
  [83] = {x=-66.93354, y=-18.726319, z=97.995995, rx=179.999705, ry=-1.999735, rz=-0.000771, shoulder=lefty, elbow=epositive, wrist=wpositive, fatherId=frmaster[2]}
  [84] = {x=-66.933761, y=-19.709039, z=97.990938, rx=-179.99895, ry=-1.999647, rz=-0.000657, shoulder=lefty, elbow=epositive, wrist=wpositive, fatherId=frmaster[2]}
  [85] = {x=-66.935051, y=-20.695687, z=97.990541, rx=-179.999691, ry=-2.000291, rz=0.000079, shoulder=lefty, elbow=epositive, wrist=wpositive, fatherId=frmaster[2]}
  [86] = {x=-66.935728, y=-21.680348, z=97.989677, rx=-179.999341, ry=-2.000098, rz=0.000227, shoulder=lefty, elbow=epositive, wrist=wpositive, fatherId=frmaster[2]}
  [87] = {x=-66.936485, y=-22.667345, z=97.993434, rx=-179.999985, ry=-1.999807, rz=0.000387, shoulder=lefty, elbow=epositive, wrist=wpositive, fatherId=frmaster[2]}
  [88] = {x=-66.937785, y=-23.652237, z=97.99675, rx=-179.999634, ry=-1.999609, rz=0.000602, shoulder=lefty, elbow=epositive, wrist=wpositive, fatherId=frmaster[2]}
  [89] = {x=-66.940293, y=-24.640475, z=97.99558, rx=179.999629, ry=-2.000238, rz=0.000458, shoulder=lefty, elbow=epositive, wrist=wpositive, fatherId=frmaster[2]}
  [90] = {x=-66.933369, y=-25.622117, z=97.997876, rx=179.999957, ry=-2.000023, rz=-0.000285, shoulder=lefty, elbow=epositive, wrist=wpositive, fatherId=frmaster[2]}
  [91] = {x=-66.935494, y=-26.609658, z=97.991594, rx=-179.999689, ry=-1.999801, rz=-0.000007, shoulder=lefty, elbow=epositive, wrist=wpositive, fatherId=frmaster[2]}
  [92] = {x=-66.938118, y=-27.594669, z=97.993964, rx=-179.999334, ry=-1.999579, rz=0.000316, shoulder=lefty, elbow=epositive, wrist=wpositive, fatherId=frmaster[2]}
  [93] = {x=-66.941923, y=-28.582536, z=98.000947, rx=179.998937, ry=-2.000099, rz=0.000284, shoulder=lefty, elbow=epositive, wrist=wpositive, fatherId=frmaster[2]}
  [94] = {x=-66.910509, y=-27.594197, z=97.989634, rx=-179.999412, ry=-1.999576, rz=0.000315, shoulder=lefty, elbow=epositive, wrist=wpositive, fatherId=frmaster[2]}
  [95] = {x=-66.889202, y=-26.611762, z=97.997302, rx=179.999183, ry=-1.999714, rz=0.000008, shoulder=lefty, elbow=epositive, wrist=wpositive, fatherId=frmaster[2]}
  [96] = {x=-66.859854, y=-25.622553, z=97.990127, rx=-179.999259, ry=-2.000123, rz=-0.000228, shoulder=lefty, elbow=epositive, wrist=wpositive, fatherId=frmaster[2]}
  [97] = {x=-66.839403, y=-24.639439, z=98.00185, rx=179.999338, ry=-2.000253, rz=-0.000469, shoulder=lefty, elbow=epositive, wrist=wpositive, fatherId=frmaster[2]}
  [98] = {x=-66.809748, y=-23.650806, z=97.989622, rx=-179.999007, ry=-1.999712, rz=-0.000319, shoulder=lefty, elbow=epositive, wrist=wpositive, fatherId=frmaster[2]}
  [99] = {x=-66.790069, y=-22.668684, z=97.996325, rx=179.999592, ry=-1.999826, rz=0.000483, shoulder=lefty, elbow=epositive, wrist=wpositive, fatherId=frmaster[2]}
  [100] = {x=-66.762302, y=-21.680258, z=97.997428, rx=-179.999843, ry=-2.000124, rz=-0.000653, shoulder=lefty, elbow=epositive, wrist=wpositive, fatherId=frmaster[2]}
  [101] = {x=-66.743802, y=-20.695288, z=97.994145, rx=-179.999251, ry=-2.000416, rz=0.000233, shoulder=lefty, elbow=epositive, wrist=wpositive, fatherId=frmaster[2]}
  [102] = {x=-66.715185, y=-19.712779, z=97.995384, rx=179.99942, ry=-1.999576, rz=0.000452, shoulder=lefty, elbow=epositive, wrist=wpositive, fatherId=frmaster[2]}
  [103] = {x=-66.688775, y=-18.724302, z=97.991221, rx=-179.999017, ry=-1.999957, rz=-0.000586, shoulder=lefty, elbow=epositive, wrist=wpositive, fatherId=frmaster[2]}
  [104] = {x=-66.662302, y=-17.739834, z=98.000731, rx=179.99956, ry=-2.000044, rz=-0.000655, shoulder=lefty, elbow=epositive, wrist=wpositive, fatherId=frmaster[2]}
  [105] = {x=-66.645316, y=-16.756157, z=98.000899, rx=179.999159, ry=-2.000218, rz=0.000306, shoulder=lefty, elbow=epositive, wrist=wpositive, fatherId=frmaster[2]}
  [106] = {x=-66.618831, y=-15.769794, z=98.000588, rx=179.999825, ry=-1.999562, rz=0.000689, shoulder=lefty, elbow=epositive, wrist=wpositive, fatherId=frmaster[2]}
  [107] = {x=-66.593804, y=-14.784654, z=97.999959, rx=179.9994, ry=-1.999725, rz=0.000693, shoulder=lefty, elbow=epositive, wrist=wpositive, fatherId=frmaster[2]}
  [108] = {x=-66.569345, y=-13.798288, z=97.998993, rx=179.999971, ry=-1.999985, rz=0.000751, shoulder=lefty, elbow=epositive, wrist=wpositive, fatherId=frmaster[2]}
  [109] = {x=-66.545194, y=-12.813219, z=97.997695, rx=179.999548, ry=-2.000136, rz=-0.000204, shoulder=lefty, elbow=epositive, wrist=wpositive, fatherId=frmaster[2]}
  [110] = {x=-66.521594, y=-11.827113, z=97.996087, rx=-179.99988, ry=-2.000386, rz=-0.000104, shoulder=lefty, elbow=epositive, wrist=wpositive, fatherId=frmaster[2]}
  [111] = {x=-66.488326, y=-10.841223, z=97.994059, rx=179.999768, ry=-1.999605, rz=-0.000638, shoulder=lefty, elbow=epositive, wrist=wpositive, fatherId=frmaster[2]}
  [112] = {x=-66.465488, y=-9.855808, z=98.000746, rx=179.999346, ry=-1.999754, rz=-0.000502, shoulder=lefty, elbow=epositive, wrist=wpositive, fatherId=frmaster[2]}
  [113] = {x=-66.44313, y=-8.870795, z=97.998257, rx=179.999921, ry=-1.999992, rz=-0.000337, shoulder=lefty, elbow=epositive, wrist=wpositive, fatherId=frmaster[2]}
  [114] = {x=-66.42139, y=-7.884239, z=97.99052, rx=-179.999503, ry=-2.000215, rz=-0.000178, shoulder=lefty, elbow=epositive, wrist=wpositive, fatherId=frmaster[2]}
  [115] = {x=-66.39096, y=-6.899301, z=97.996285, rx=-179.99995, ry=-2.000349, rz=-0.000981, shoulder=lefty, elbow=epositive, wrist=wpositive, fatherId=frmaster[2]}
  [116] = {x=-66.368797, y=-5.91401, z=97.996843, rx=179.999729, ry=-1.999555, rz=0.000606, shoulder=lefty, elbow=epositive, wrist=wpositive, fatherId=frmaster[2]}
  [117] = {x=-66.34812, y=-4.92963, z=97.997195, rx=179.999311, ry=-1.999673, rz=0.000822, shoulder=lefty, elbow=epositive, wrist=wpositive, fatherId=frmaster[2]}
  [118] = {x=-66.319584, y=-3.940403, z=97.992289, rx=-179.999142, ry=-1.999989, rz=0.000102, shoulder=lefty, elbow=epositive, wrist=wpositive, fatherId=frmaster[2]}
  [119] = {x=-66.290859, y=-2.95676, z=98.00089, rx=179.999418, ry=-2.000003, rz=-0.000649, shoulder=lefty, elbow=epositive, wrist=wpositive, fatherId=frmaster[2]}
  [120] = {x=-66.271634, y=-1.971891, z=97.995631, rx=179.999998, ry=-2.000208, rz=-0.000361, shoulder=lefty, elbow=epositive, wrist=wpositive, fatherId=frmaster[2]}
  [121] = {x=-66.244376, y=-0.983641, z=97.99391, rx=-179.999449, ry=-2.000409, rz=-0.000053, shoulder=lefty, elbow=epositive, wrist=wpositive, fatherId=frmaster[2]}
  [122] = {x=-66.224642, y=-0.001016, z=97.99697, rx=-179.999766, ry=-1.999603, rz=0.000678, shoulder=lefty, elbow=epositive, wrist=wpositive, fatherId=frmaster[2]}
  [123] = {x=-66.197953, y=0.983563, z=97.994876, rx=179.999794, ry=-1.999692, rz=-0.000004, shoulder=lefty, elbow=epositive, wrist=wpositive, fatherId=frmaster[2]}
  [124] = {x=-66.172041, y=1.971387, z=97.996381, rx=-179.999652, ry=-1.999888, rz=0.000371, shoulder=lefty, elbow=epositive, wrist=wpositive, fatherId=frmaster[2]}
  [125] = {x=-66.146336, y=2.956587, z=97.997711, rx=179.999909, ry=-1.999973, rz=-0.000268, shoulder=lefty, elbow=epositive, wrist=wpositive, fatherId=frmaster[2]}
  [126] = {x=-66.121345, y=3.943753, z=97.993972, rx=-179.999535, ry=-2.000153, rz=0.000124, shoulder=lefty, elbow=epositive, wrist=wpositive, fatherId=frmaster[2]}
  [127] = {x=-66.09668, y=4.929368, z=97.990101, rx=-179.998978, ry=-2.000332, rz=-0.000464, shoulder=lefty, elbow=epositive, wrist=wpositive, fatherId=frmaster[2]}
  [128] = {x=-66.07212, y=5.912079, z=97.994719, rx=179.999589, ry=-2.000303, rz=-0.000073, shoulder=lefty, elbow=epositive, wrist=wpositive, fatherId=frmaster[2]}
  [129] = {x=-66.047289, y=6.897906, z=97.99427, rx=-179.999754, ry=-1.999578, rz=-0.000193, shoulder=lefty, elbow=epositive, wrist=wpositive, fatherId=frmaster[2]}
  [130] = {x=-66.024039, y=7.884074, z=97.99743, rx=179.99981, ry=-1.999644, rz=0.000252, shoulder=lefty, elbow=epositive, wrist=wpositive, fatherId=frmaster[2]}
  [131] = {x=-66.001086, y=8.868411, z=98.000467, rx=179.999374, ry=-1.99971, rz=0.000719, shoulder=lefty, elbow=epositive, wrist=wpositive, fatherId=frmaster[2]}
  [132] = {x=-65.970344, y=9.855529, z=97.998446, rx=179.999907, ry=-1.999872, rz=-0.000786, shoulder=lefty, elbow=epositive, wrist=wpositive, fatherId=frmaster[2]}
  [133] = {x=-65.948632, y=10.841847, z=97.991535, rx=-179.999533, ry=-2.000024, rz=-0.000294, shoulder=lefty, elbow=epositive, wrist=wpositive, fatherId=frmaster[2]}
  [134] = {x=-65.92712, y=11.826085, z=97.993077, rx=-179.999967, ry=-2.000075, rz=0.000212, shoulder=lefty, elbow=epositive, wrist=wpositive, fatherId=frmaster[2]}
  [135] = {x=-65.897777, y=12.812894, z=97.998102, rx=179.999572, ry=-2.000125, rz=-0.000262, shoulder=lefty, elbow=epositive, wrist=wpositive, fatherId=frmaster[2]}
  [136] = {x=-65.877212, y=13.796438, z=97.994633, rx=-179.999866, ry=-2.000276, rz=0.000295, shoulder=lefty, elbow=epositive, wrist=wpositive, fatherId=frmaster[2]}
  [137] = {x=-65.849106, y=14.784817, z=97.98981, rx=-179.99933, ry=-2.000414, rz=-0.000152, shoulder=lefty, elbow=epositive, wrist=wpositive, fatherId=frmaster[2]}
  [138] = {x=-65.828084, y=15.766236, z=97.99827, rx=179.999344, ry=-1.999461, rz=0.000849, shoulder=lefty, elbow=epositive, wrist=wpositive, fatherId=frmaster[2]}
  [139] = {x=-65.800853, y=16.75355, z=97.996951, rx=179.999881, ry=-1.999601, rz=0.000447, shoulder=lefty, elbow=epositive, wrist=wpositive, fatherId=frmaster[2]}
  [140] = {x=-65.774163, y=17.740875, z=97.990764, rx=-179.999581, ry=-1.999728, rz=0.000041, shoulder=lefty, elbow=epositive, wrist=wpositive, fatherId=frmaster[2]}
  [141] = {x=-65.747663, y=18.725693, z=97.992963, rx=179.999962, ry=-1.999756, rz=-0.000351, shoulder=lefty, elbow=epositive, wrist=wpositive, fatherId=frmaster[2]}
  [142] = {x=-65.730055, y=19.71041, z=97.99876, rx=179.999532, ry=-1.999786, rz=0.000279, shoulder=lefty, elbow=epositive, wrist=wpositive, fatherId=frmaster[2]}
  [143] = {x=-65.704873, y=20.697423, z=97.991278, rx=-179.998935, ry=-2.000019, rz=-0.000053, shoulder=lefty, elbow=epositive, wrist=wpositive, fatherId=frmaster[2]}
  [144] = {x=-65.679643, y=21.68048, z=98.000498, rx=179.999615, ry=-1.999935, rz=0.000586, shoulder=lefty, elbow=epositive, wrist=wpositive, fatherId=frmaster[2]}
  [145] = {x=-65.655422, y=22.667028, z=97.991752, rx=-179.999845, ry=-2.000043, rz=0.000237, shoulder=lefty, elbow=epositive, wrist=wpositive, fatherId=frmaster[2]}
  [146] = {x=-65.631423, y=23.651944, z=97.999667, rx=179.9997, ry=-2.000064, rz=-0.000071, shoulder=lefty, elbow=epositive, wrist=wpositive, fatherId=frmaster[2]}
  [147] = {x=-65.599793, y=24.637759, z=97.994412, rx=-179.999785, ry=-2.000174, rz=-0.000376, shoulder=lefty, elbow=epositive, wrist=wpositive, fatherId=frmaster[2]}
  [148] = {x=-65.577168, y=25.625642, z=97.99624, rx=179.999762, ry=-2.000172, rz=-0.000693, shoulder=lefty, elbow=epositive, wrist=wpositive, fatherId=frmaster[2]}
  [149] = {x=-65.554552, y=26.608184, z=97.994617, rx=-179.999697, ry=-2.000288, rz=0.000048, shoulder=lefty, elbow=epositive, wrist=wpositive, fatherId=frmaster[2]}
  [150] = {x=-65.53256, y=27.592668, z=97.999963, rx=179.998856, ry=-2.000172, rz=-0.000259, shoulder=lefty, elbow=epositive, wrist=wpositive, fatherId=frmaster[2]}
  [151] = {x=-65.503198, y=28.580264, z=98.000497, rx=179.999372, ry=-2.000278, rz=-0.000501, shoulder=lefty, elbow=epositive, wrist=wpositive, fatherId=frmaster[2]}
  [152] = {x=-65.838163, y=27.84263, z=98.187395, rx=-179.101306, ry=-1.787196, rz=0.013692, shoulder=lefty, elbow=epositive, wrist=wpositive, fatherId=frmaster[2]}
  [153] = {x=-66.479353, y=27.725374, z=98.008437, rx=-178.574399, ry=-1.402056, rz=0.017937, shoulder=lefty, elbow=epositive, wrist=wpositive, fatherId=frmaster[2]}
  [154] = {x=-66.594932, y=27.112453, z=97.572839, rx=-178.203772, ry=-0.879237, rz=0.013602, shoulder=lefty, elbow=epositive, wrist=wpositive, fatherId=frmaster[2]}
  [155] = {x=-67.312864, y=26.791648, z=96.64441, rx=-178.000264, ry=0.000237, rz=-0.000733, shoulder=lefty, elbow=epositive, wrist=wpositive, fatherId=frmaster[2]}
  [156] = {x=-66.323261, y=26.802148, z=96.645277, rx=-177.999899, ry=0.000009, rz=0.000865, shoulder=lefty, elbow=epositive, wrist=wpositive, fatherId=frmaster[2]}
  [157] = {x=-65.324808, y=26.811115, z=96.642512, rx=-178.000515, ry=-0.00016, rz=0.000461, shoulder=lefty, elbow=epositive, wrist=wpositive, fatherId=frmaster[2]}
  [158] = {x=-64.326337, y=26.8247, z=96.639813, rx=-177.999131, ry=-0.000512, rz=0.000055, shoulder=lefty, elbow=epositive, wrist=wpositive, fatherId=frmaster[2]}
  [159] = {x=-63.325997, y=26.835652, z=96.641805, rx=-177.999644, ry=0.000229, rz=0.000068, shoulder=lefty, elbow=epositive, wrist=wpositive, fatherId=frmaster[2]}
  [160] = {x=-62.326274, y=26.846278, z=96.64031, rx=-177.999238, ry=-0.00002, rz=-0.000355, shoulder=lefty, elbow=epositive, wrist=wpositive, fatherId=frmaster[2]}
  [161] = {x=-61.334472, y=26.857859, z=96.638863, rx=-177.998834, ry=-0.000233, rz=0.000219, shoulder=lefty, elbow=epositive, wrist=wpositive, fatherId=frmaster[2]}
  [162] = {x=-60.333357, y=26.865458, z=96.646829, rx=-178.000402, ry=-0.000262, rz=-0.000233, shoulder=lefty, elbow=epositive, wrist=wpositive, fatherId=frmaster[2]}
  [163] = {x=-59.339579, y=26.877884, z=96.641834, rx=-177.999888, ry=0.000428, rz=0.000769, shoulder=lefty, elbow=epositive, wrist=wpositive, fatherId=frmaster[2]}
  [164] = {x=-58.337678, y=26.88748, z=96.64629, rx=-178.000443, ry=0.000307, rz=-0.000689, shoulder=lefty, elbow=epositive, wrist=wpositive, fatherId=frmaster[2]}
  [165] = {x=-57.343757, y=26.898058, z=96.642525, rx=-178.000006, ry=0.000112, rz=-0.000137, shoulder=lefty, elbow=epositive, wrist=wpositive, fatherId=frmaster[2]}
  [166] = {x=-56.349093, y=26.907126, z=96.643488, rx=-178.000554, ry=0.000034, rz=0.0004, shoulder=lefty, elbow=epositive, wrist=wpositive, fatherId=frmaster[2]}
  [167] = {x=-55.346114, y=26.920944, z=96.644402, rx=-178.000092, ry=-0.000185, rz=-0.000066, shoulder=lefty, elbow=epositive, wrist=wpositive, fatherId=frmaster[2]}
  [168] = {x=-54.35063, y=26.932011, z=96.64184, rx=-177.999631, ry=-0.000369, rz=-0.000534, shoulder=lefty, elbow=epositive, wrist=wpositive, fatherId=frmaster[2]}
  [169] = {x=-53.354371, y=26.941589, z=96.644007, rx=-178.000154, ry=-0.000428, rz=-0.000018, shoulder=lefty, elbow=epositive, wrist=wpositive, fatherId=frmaster[2]}
  [170] = {x=-52.356449, y=26.951108, z=96.642671, rx=-177.99957, ry=0.000295, rz=-0.000074, shoulder=lefty, elbow=epositive, wrist=wpositive, fatherId=frmaster[2]}
  [171] = {x=-51.359182, y=26.961495, z=96.64126, rx=-178.000075, ry=0.000244, rz=0.000436, shoulder=lefty, elbow=epositive, wrist=wpositive, fatherId=frmaster[2]}
  [172] = {x=-50.361253, y=26.971628, z=96.644622, rx=-178.000572, ry=0.000205, rz=-0.000069, shoulder=lefty, elbow=epositive, wrist=wpositive, fatherId=frmaster[2]}
  [173] = {x=-49.36326, y=26.985266, z=96.639708, rx=-177.999077, ry=-0.000086, rz=-0.000564, shoulder=lefty, elbow=epositive, wrist=wpositive, fatherId=frmaster[2]}
  [174] = {x=-48.372463, y=26.99477, z=96.63955, rx=-177.999566, ry=-0.000085, rz=0.000925, shoulder=lefty, elbow=epositive, wrist=wpositive, fatherId=frmaster[2]}
  [175] = {x=-47.372808, y=27.005494, z=96.644099, rx=-178.000038, ry=-0.000106, rz=0.000398, shoulder=lefty, elbow=epositive, wrist=wpositive, fatherId=frmaster[2]}
  [176] = {x=-46.372378, y=27.01486, z=96.645082, rx=-178.000501, ry=-0.000123, rz=-0.000132, shoulder=lefty, elbow=epositive, wrist=wpositive, fatherId=frmaster[2]}
  [177] = {x=-45.379969, y=27.026155, z=96.646144, rx=-177.999973, ry=-0.000233, rz=0.000334, shoulder=lefty, elbow=epositive, wrist=wpositive, fatherId=frmaster[2]}
  [178] = {x=-44.378434, y=27.0364, z=96.643522, rx=-178.00042, ry=-0.000241, rz=-0.000201, shoulder=lefty, elbow=epositive, wrist=wpositive, fatherId=frmaster[2]}
  [179] = {x=-43.384348, y=27.04489, z=96.645742, rx=-178.000866, ry=-0.000204, rz=0.000246, shoulder=lefty, elbow=epositive, wrist=wpositive, fatherId=frmaster[2]}
  [180] = {x=-42.381937, y=27.058382, z=96.647902, rx=-178.000305, ry=-0.000334, rz=-0.00031, shoulder=lefty, elbow=epositive, wrist=wpositive, fatherId=frmaster[2]}
  [181] = {x=-41.386708, y=27.067756, z=96.646508, rx=-178.000734, ry=-0.000289, rz=0.000131, shoulder=lefty, elbow=epositive, wrist=wpositive, fatherId=frmaster[2]}
  [182] = {x=-40.390733, y=27.07692, z=96.649888, rx=-178.001154, ry=-0.000232, rz=-0.000444, shoulder=lefty, elbow=epositive, wrist=wpositive, fatherId=frmaster[2]}
  [183] = {x=-39.394508, y=27.088395, z=96.64491, rx=-178.000577, ry=-0.000321, rz=-0.00001, shoulder=lefty, elbow=epositive, wrist=wpositive, fatherId=frmaster[2]}
  [184] = {x=-38.39753, y=27.099674, z=96.644705, rx=-177.999991, ry=-0.000403, rz=0.000408, shoulder=lefty, elbow=epositive, wrist=wpositive, fatherId=frmaster[2]}
  [185] = {x=-37.399425, y=27.108355, z=96.649191, rx=-178.001373, ry=-0.00018, rz=-0.000191, shoulder=lefty, elbow=epositive, wrist=wpositive, fatherId=frmaster[2]}
  [186] = {x=-36.401427, y=27.121776, z=96.645392, rx=-177.999782, ry=-0.000407, rz=0.00022, shoulder=lefty, elbow=epositive, wrist=wpositive, fatherId=frmaster[2]}
  [187] = {x=-35.402285, y=27.132614, z=96.646283, rx=-178.000159, ry=-0.000325, rz=-0.000386, shoulder=lefty, elbow=epositive, wrist=wpositive, fatherId=frmaster[2]}
  [188] = {x=-34.410417, y=27.14045, z=96.643638, rx=-178.000535, ry=-0.000203, rz=0.000004, shoulder=lefty, elbow=epositive, wrist=wpositive, fatherId=frmaster[2]}
  [189] = {x=-33.41022, y=27.153456, z=96.64092, rx=-177.999907, ry=-0.000268, rz=0.000392, shoulder=lefty, elbow=epositive, wrist=wpositive, fatherId=frmaster[2]}
  [190] = {x=-32.409032, y=27.165114, z=96.642936, rx=-178.000257, ry=-0.000167, rz=-0.000239, shoulder=lefty, elbow=epositive, wrist=wpositive, fatherId=frmaster[2]}
  [191] = {x=-31.415287, y=27.174949, z=96.641449, rx=-177.99962, ry=-0.000188, rz=0.000127, shoulder=lefty, elbow=epositive, wrist=wpositive, fatherId=frmaster[2]}
  [192] = {x=-30.420524, y=27.183424, z=96.644696, rx=-177.99996, ry=-0.000038, rz=0.000475, shoulder=lefty, elbow=epositive, wrist=wpositive, fatherId=frmaster[2]}
  [193] = {x=-29.417231, y=27.19596, z=96.647829, rx=-178.000282, ry=0.000082, rz=-0.00018, shoulder=lefty, elbow=epositive, wrist=wpositive, fatherId=frmaster[2]}
  [194] = {x=-28.421155, y=27.205444, z=96.647408, rx=-178.000605, ry=0.000242, rz=0.00016, shoulder=lefty, elbow=epositive, wrist=wpositive, fatherId=frmaster[2]}
  [195] = {x=-27.425006, y=27.218475, z=96.638615, rx=-177.998948, ry=0.000061, rz=0.000512, shoulder=lefty, elbow=epositive, wrist=wpositive, fatherId=frmaster[2]}
  [196] = {x=-26.427035, y=27.226511, z=96.647705, rx=-178.000236, ry=0.00041, rz=-0.000184, shoulder=lefty, elbow=epositive, wrist=wpositive, fatherId=frmaster[2]}
  [197] = {x=-25.429863, y=27.236716, z=96.648372, rx=-178.000688, ry=-0.000306, rz=-0.000289, shoulder=lefty, elbow=epositive, wrist=wpositive, fatherId=frmaster[2]}
  [198] = {x=-24.431312, y=27.249472, z=96.640619, rx=-177.999992, ry=-0.000305, rz=0.000037, shoulder=lefty, elbow=epositive, wrist=wpositive, fatherId=frmaster[2]}
  [199] = {x=-23.439357, y=27.256646, z=96.642496, rx=-178.000278, ry=-0.00008, rz=0.00033, shoulder=lefty, elbow=epositive, wrist=wpositive, fatherId=frmaster[2]}
  [200] = {x=-22.438851, y=27.268013, z=96.64425, rx=-178.000546, ry=0.000117, rz=-0.000381, shoulder=lefty, elbow=epositive, wrist=wpositive, fatherId=frmaster[2]}
  [201] = {x=-21.43819, y=27.28289, z=96.645991, rx=-177.999822, ry=0.000137, rz=-0.000095, shoulder=lefty, elbow=epositive, wrist=wpositive, fatherId=frmaster[2]}
